C09129=1122.210,43.418,-53.082,179.810,7.126,149.381
C09130=1122.214,43.168,-53.066,179.809,7.121,149.380
C09131=1122.220,42.919,-53.051,179.808,7.117,149.380
C09132=1122.225,42.670,-53.035,179.807,7.113,149.379
C09133=1122.230,42.420,-53.019,179.806,7.109,149.379
C09134=1122.235,42.170,-53.004,179.805,7.105,149.378
C09135=1122.240,41.921,-52.989,179.804,7.101,149.377
C09136=1122.245,41.672,-52.973,179.803,7.097,149.377
C09137=1122.250,41.422,-52.956,179.802,7.093,149.376
C09138=1122.255,41.173,-52.941,179.800,7.088,149.376
C09139=1122.260,40.924,-52.926,179.799,7.084,149.375
C09140=1122.264,40.674,-52.910,179.798,7.080,149.374
C09141=1122.270,40.424,-52.894,179.797,7.076,149.374
C09142=1122.275,40.175,-52.879,179.796,7.072,149.373
C09143=1122.280,39.926,-52.864,179.795,7.067,149.373
C09144=1122.285,39.676,-52.848,179.794,7.063,149.372
C09145=1122.290,39.426,-52.832,179.792,7.059,149.371
C09146=1122.295,39.177,-52.817,179.791,7.055,149.371
C09147=1122.300,38.928,-52.802,179.790,7.050,149.370
C09148=1122.305,38.678,-52.786,179.789,7.046,149.369
C09149=1122.310,38.428,-52.771,179.788,7.042,149.369
C09150=1122.315,38.179,-52.755,179.786,7.038,149.368
C09151=1122.320,37.930,-52.739,179.785,7.034,149.368
C09152=1122.325,37.681,-52.724,179.784,7.029,149.367
C09153=1122.330,37.430,-52.708,179.783,7.025,149.366
C09154=1122.335,37.181,-52.693,179.783,7.021,149.366
C09155=1122.340,36.932,-52.678,179.781,7.018,149.365
C09156=1122.345,36.682,-52.663,179.780,7.013,149.365
C09157=1122.350,36.433,-52.648,179.779,7.009,149.364
C09158=1122.356,36.183,-52.632,179.778,7.005,149.363
C09159=1122.360,35.933,-52.616,179.777,7.000,149.363
C09160=1122.365,35.684,-52.601,179.776,6.996,149.362
C09161=1122.370,35.469,-52.588,179.774,6.992,149.362
C09162=1122.374,35.254,-52.575,179.774,6.989,149.361
C09163=1122.378,35.040,-52.562,179.773,6.985,149.361
C09164=1122.383,34.825,-52.549,179.772,6.981,149.360
C09165=1122.387,34.609,-52.535,179.771,6.978,149.360
C09166=1122.391,34.395,-52.523,179.770,6.974,149.359
C09167=1122.395,34.180,-52.509,179.769,6.970,149.358
C09168=1122.400,33.966,-52.496,179.768,6.966,149.358
C09169=1122.405,33.716,-52.481,179.767,6.962,149.357
C09170=1122.410,33.466,-52.466,179.766,6.958,149.357
C09171=1122.416,33.217,-52.451,179.765,6.954,149.356
C09172=1122.420,32.967,-52.436,179.764,6.950,149.355
C09173=1122.425,32.718,-52.420,179.763,6.946,149.355
C09174=1122.430,32.468,-52.406,179.762,6.941,149.354
C09175=1122.435,32.219,-52.390,179.760,6.937,149.353
C09176=1122.440,31.970,-52.375,179.759,6.933,149.353
C09177=1122.446,31.720,-52.360,179.758,6.929,149.352
C09178=1122.450,31.470,-52.345,179.757,6.924,149.352
C09179=1122.455,31.221,-52.330,179.756,6.920,149.351
C09180=1122.461,30.971,-52.315,179.755,6.916,149.350
C09181=1122.465,30.722,-52.300,179.754,6.911,149.350
C09182=1122.470,30.472,-52.284,179.753,6.907,149.349
C09183=1122.475,30.222,-52.270,179.752,6.903,149.348
C09184=1122.480,29.973,-52.255,179.751,6.898,149.348
C09185=1122.485,29.724,-52.240,179.750,6.894,149.347
C09186=1122.490,29.474,-52.225,179.749,6.890,149.346
C09187=1122.495,29.225,-52.210,179.748,6.885,149.346
C09188=1122.500,28.975,-52.195,179.747,6.881,149.345
C09189=1122.506,28.726,-52.180,179.746,6.876,149.344
C09190=1122.511,28.476,-52.166,179.745,6.872,149.344
C09191=1122.515,28.227,-52.151,179.744,6.868,149.343
C09192=1122.521,27.978,-52.135,179.743,6.863,149.342
C09193=1122.526,27.728,-52.121,179.742,6.859,149.342
C09194=1122.530,27.479,-52.106,179.741,6.855,149.341
C09195=1122.536,27.229,-52.091,179.740,6.850,149.340
C09196=1122.541,26.980,-52.076,179.739,6.846,149.340
C09197=1122.546,26.730,-52.062,179.738,6.842,149.339
C09198=1122.551,26.481,-52.046,179.737,6.838,149.338
C09199=1122.556,26.231,-52.032,179.736,6.833,149.337
C09200=1122.561,25.981,-52.017,179.735,6.829,149.337
C09201=1122.566,25.732,-52.002,179.734,6.824,149.336
C09202=1122.571,25.482,-51.988,179.733,6.820,149.335
C09203=1122.576,25.233,-51.973,179.732,6.816,149.335
C09204=1122.581,24.983,-51.958,179.731,6.811,149.334
C09205=1122.586,24.734,-51.943,179.730,6.807,149.334
C09206=1122.591,24.484,-51.928,179.729,6.802,149.333
C09207=1122.596,24.234,-51.914,179.728,6.798,149.332
C09208=1122.602,23.985,-51.899,179.727,6.794,149.331
C09209=1122.607,23.735,-51.884,179.726,6.789,149.331
C09210=1122.611,23.486,-51.870,179.725,6.785,149.330
C09211=1122.617,23.237,-51.855,179.724,6.780,149.329
C09212=1122.622,22.987,-51.841,179.723,6.776,149.329
C09213=1122.627,22.737,-51.826,179.722,6.772,149.328
C09214=1122.632,22.488,-51.811,179.721,6.767,149.327
C09215=1122.637,22.239,-51.797,179.721,6.763,149.326
C09216=1122.642,21.989,-51.783,179.720,6.758,149.326
C09217=1122.647,21.774,-51.770,179.719,6.754,149.325
C09218=1122.650,21.559,-51.757,179.718,6.751,149.325
C09219=1122.655,21.344,-51.745,179.717,6.747,149.324
C09220=1122.659,21.129,-51.733,179.716,6.743,149.323
C09221=1122.664,20.914,-51.720,179.715,6.739,149.323
C09222=1122.668,20.699,-51.707,179.715,6.735,149.322
C09223=1122.673,20.484,-51.695,179.714,6.731,149.321
C09224=1122.676,20.269,-51.683,179.713,6.728,149.321
C09225=1122.682,20.019,-51.668,179.712,6.723,149.320
C09226=1122.687,19.770,-51.653,179.711,6.719,149.319
C09227=1122.692,19.521,-51.639,179.710,6.714,149.319
C09228=1122.697,19.271,-51.624,179.710,6.710,149.318
C09229=1122.702,19.022,-51.610,179.709,6.705,149.317
C09230=1122.707,18.772,-51.596,179.707,6.700,149.317
C09231=1122.712,18.522,-51.582,179.706,6.695,149.316
C09232=1122.717,18.273,-51.567,179.705,6.691,149.315
C09233=1122.722,18.023,-51.553,179.705,6.686,149.314
C09234=1122.727,17.775,-51.538,179.704,6.682,149.313
C09235=1122.733,17.524,-51.524,179.703,6.678,149.313
C09236=1122.738,17.275,-51.509,179.702,6.673,149.312
C09237=1122.743,17.025,-51.495,179.701,6.669,149.311
C09238=1122.748,16.775,-51.481,179.700,6.664,149.310
C09239=1122.753,16.526,-51.467,179.699,6.660,149.310
C09240=1122.758,16.277,-51.453,179.698,6.655,149.309
C09241=1122.763,16.027,-51.438,179.698,6.651,149.308
C09242=1122.768,15.777,-51.424,179.697,6.646,149.308
C09243=1122.773,15.527,-51.410,179.696,6.642,149.307
C09244=1122.779,15.278,-51.396,179.695,6.637,149.306
C09245=1122.784,15.029,-51.382,179.695,6.633,149.305
C09246=1122.789,14.779,-51.367,179.693,6.628,149.305
C09247=1122.794,14.529,-51.353,179.692,6.623,149.304
C09248=1122.799,14.280,-51.339,179.691,6.618,149.303
C09249=1122.804,14.031,-51.325,179.691,6.614,149.302
C09250=1122.809,13.781,-51.311,179.690,6.609,149.301
C09251=1122.813,13.532,-51.297,179.689,6.605,149.301
C09252=1122.819,13.283,-51.283,179.688,6.600,149.300
C09253=1122.824,13.033,-51.269,179.688,6.596,149.299
C09254=1122.829,12.783,-51.254,179.687,6.591,149.298
C09255=1122.834,12.533,-51.240,179.686,6.587,149.298
C09256=1122.840,12.284,-51.227,179.686,6.582,149.297
C09257=1122.845,12.034,-51.213,179.684,6.577,149.296
C09258=1122.850,11.784,-51.198,179.683,6.572,149.295
C09259=1122.855,11.535,-51.184,179.682,6.568,149.294
C09260=1122.860,11.286,-51.170,179.682,6.563,149.294
C09261=1122.865,11.036,-51.156,179.681,6.558,149.293
C09262=1122.870,10.787,-51.143,179.680,6.554,149.292
C09263=1122.875,10.537,-51.129,179.680,6.549,149.291
C09264=1122.880,10.287,-51.115,179.679,6.545,149.291
C09265=1122.885,10.037,-51.100,179.678,6.540,149.290
C09266=1122.891,9.788,-51.087,179.678,6.536,149.289
C09267=1122.895,9.539,-51.072,179.676,6.530,149.288
C09268=1122.900,9.289,-51.059,179.675,6.526,149.287
C09269=1122.906,9.040,-51.045,179.675,6.521,149.286
C09270=1122.911,8.790,-51.031,179.674,6.516,149.286
C09271=1122.916,8.541,-51.017,179.673,6.512,149.285
C09272=1122.921,8.291,-51.004,179.673,6.507,149.284
C09273=1122.925,8.076,-50.991,179.672,6.504,149.283
C09274=1122.929,7.861,-50.980,179.672,6.499,149.282
C09275=1122.934,7.645,-50.968,179.671,6.495,149.282
C09276=1122.939,7.431,-50.956,179.671,6.492,149.281
C09277=1122.943,7.215,-50.944,179.670,6.487,149.280
C09278=1122.947,7.000,-50.933,179.670,6.484,149.280
C09279=1122.951,6.785,-50.920,179.670,6.480,149.279
C09280=1122.956,6.571,-50.909,179.670,6.476,149.278
C09281=1122.961,6.321,-50.895,179.669,6.471,149.277
C09282=1122.966,6.071,-50.881,179.669,6.467,149.276
C09283=1122.972,5.822,-50.867,179.668,6.462,149.275
C09284=1122.976,5.572,-50.854,179.667,6.458,149.275
C09285=1122.982,5.323,-50.840,179.667,6.454,149.274
C09286=1122.987,5.073,-50.826,179.667,6.449,149.273
C09287=1122.992,4.823,-50.812,179.666,6.444,149.272
C09288=1122.997,4.574,-50.799,179.665,6.440,149.271
C09289=1123.002,4.324,-50.786,179.665,6.435,149.270
C09290=1123.008,4.075,-50.772,179.664,6.430,149.269
C09291=1123.012,3.825,-50.758,179.664,6.427,149.269
C09292=1123.018,3.576,-50.745,179.663,6.422,149.268
C09293=1123.023,3.326,-50.730,179.663,6.417,149.267
C09294=1123.027,3.076,-50.718,179.662,6.412,149.266
C09295=1123.033,2.827,-50.704,179.662,6.408,149.265
C09296=1123.038,2.577,-50.690,179.661,6.404,149.265
C09297=1123.043,2.328,-50.677,179.661,6.400,149.264
C09298=1123.048,2.078,-50.663,179.660,6.395,149.263
C09299=1123.054,1.829,-50.649,179.660,6.390,149.262
C09300=1123.058,1.579,-50.636,179.659,6.385,149.261
C09301=1123.064,1.330,-50.622,179.658,6.381,149.260
C09302=1123.068,1.080,-50.609,179.658,6.377,149.260
C09303=1123.074,0.831,-50.595,179.658,6.372,149.259
C09304=1123.079,0.580,-50.582,179.657,6.368,149.258
C09305=1123.084,0.331,-50.569,179.656,6.363,149.257
C09306=1123.089,0.081,-50.555,179.656,6.359,149.256
C09307=1123.094,-0.168,-50.542,179.655,6.354,149.255
C09308=1123.099,-0.418,-50.528,179.655,6.349,149.254
C09309=1123.104,-0.667,-50.516,179.654,6.346,149.254
C09310=1123.110,-0.917,-50.502,179.654,6.341,149.253
C09311=1123.115,-1.166,-50.488,179.653,6.336,149.252
C09312=1123.120,-1.417,-50.475,179.652,6.332,149.251
C09313=1123.125,-1.666,-50.461,179.652,6.327,149.250
C09314=1123.130,-1.916,-50.448,179.651,6.322,149.250
C09315=1123.136,-2.165,-50.435,179.651,6.318,149.249
C09316=1123.140,-2.415,-50.421,179.650,6.314,149.248
C09317=1123.146,-2.664,-50.408,179.650,6.309,149.247
C09318=1123.150,-2.914,-50.395,179.649,6.305,149.246
C09319=1123.156,-3.163,-50.381,179.648,6.300,149.246
C09320=1123.161,-3.413,-50.369,179.648,6.296,149.245
C09321=1123.166,-3.663,-50.355,179.647,6.291,149.244
C09322=1123.171,-3.912,-50.343,179.647,6.286,149.243
C09323=1123.176,-4.162,-50.328,179.646,6.282,149.242
C09324=1123.181,-4.411,-50.316,179.645,6.277,149.241
C09325=1123.187,-4.661,-50.302,179.645,6.273,149.241
C09326=1123.192,-4.911,-50.289,179.644,6.269,149.240
C09327=1123.197,-5.160,-50.276,179.644,6.264,149.239
C09328=1123.202,-5.410,-50.263,179.643,6.259,149.238
C09329=1123.207,-5.624,-50.251,179.642,6.255,149.237
C09330=1123.211,-5.840,-50.240,179.642,6.251,149.237
C09331=1123.215,-6.056,-50.229,179.641,6.248,149.236
C09332=1123.220,-6.270,-50.217,179.640,6.244,149.235
C09333=1123.225,-6.486,-50.206,179.641,6.240,149.235
C09334=1123.229,-6.701,-50.195,179.640,6.236,149.234
C09335=1123.234,-6.916,-50.183,179.639,6.232,149.233
C09336=1123.237,-7.131,-50.172,179.639,6.228,149.233
C09337=1123.243,-7.380,-50.159,179.638,6.224,149.232
C09338=1123.248,-7.630,-50.146,179.637,6.219,149.231
C09339=1123.253,-7.880,-50.133,179.637,6.214,149.230
C09340=1123.258,-8.129,-50.120,179.636,6.210,149.229
C09341=1123.263,-8.379,-50.107,179.635,6.205,149.229
C09342=1123.269,-8.629,-50.094,179.635,6.201,149.228
C09343=1123.274,-8.878,-50.082,179.634,6.196,149.227
C09344=1123.278,-9.128,-50.069,179.633,6.192,149.226
C09345=1123.284,-9.377,-50.055,179.633,6.187,149.225
C09346=1123.289,-9.627,-50.042,179.632,6.182,149.224
C09347=1123.294,-9.877,-50.029,179.631,6.178,149.224
C09348=1123.299,-10.126,-50.016,179.631,6.173,149.223
C09349=1123.305,-10.376,-50.003,179.630,6.168,149.222
C09350=1123.310,-10.625,-49.991,179.630,6.164,149.221
C09351=1123.314,-10.875,-49.978,179.629,6.159,149.220
C09352=1123.320,-11.125,-49.965,179.628,6.155,149.219
C09353=1123.325,-11.374,-49.952,179.628,6.150,149.219
C09354=1123.330,-11.624,-49.939,179.627,6.145,149.218
C09355=1123.336,-11.874,-49.926,179.626,6.141,149.217
C09356=1123.341,-12.123,-49.913,179.626,6.136,149.216
C09357=1123.345,-12.373,-49.900,179.625,6.132,149.215
C09358=1123.350,-12.622,-49.888,179.624,6.127,149.215
C09359=1123.356,-12.872,-49.876,179.624,6.122,149.214
C09360=1123.362,-13.122,-49.863,179.623,6.118,149.213
C09361=1123.366,-13.372,-49.850,179.622,6.113,149.212
C09362=1123.371,-13.621,-49.837,179.622,6.108,149.211
C09363=1123.376,-13.870,-49.824,179.621,6.104,149.211
C09364=1123.382,-14.120,-49.811,179.620,6.099,149.210
C09365=1123.387,-14.370,-49.798,179.620,6.095,149.209
C09366=1123.392,-14.619,-49.786,179.619,6.090,149.208
C09367=1123.397,-14.869,-49.773,179.618,6.086,149.207
C09368=1123.402,-15.119,-49.761,179.618,6.081,149.206
C09369=1123.408,-15.368,-49.749,179.617,6.076,149.206
C09370=1123.413,-15.618,-49.735,179.616,6.072,149.205
C09371=1123.418,-15.868,-49.722,179.615,6.066,149.204
C09372=1123.423,-16.117,-49.710,179.615,6.061,149.203
C09373=1123.429,-16.367,-49.698,179.614,6.057,149.202
C09374=1123.434,-16.616,-49.685,179.613,6.052,149.201
C09375=1123.438,-16.866,-49.672,179.613,6.048,149.201
C09376=1123.443,-17.116,-49.660,179.612,6.043,149.200
C09377=1123.449,-17.365,-49.647,179.611,6.039,149.199
C09378=1123.455,-17.615,-49.635,179.611,6.034,149.198
C09379=1123.460,-17.864,-49.622,179.610,6.029,149.197
C09380=1123.464,-18.114,-49.609,179.609,6.024,149.197
C09381=1123.470,-18.364,-49.597,179.608,6.019,149.196
C09382=1123.475,-18.614,-49.585,179.608,6.014,149.195
C09383=1123.480,-18.863,-49.572,179.607,6.010,149.194
C09384=1123.485,-19.112,-49.559,179.606,6.005,149.193
C09385=1123.490,-19.328,-49.548,179.606,6.001,149.192
C09386=1123.494,-19.543,-49.538,179.605,5.997,149.192
C09387=1123.499,-19.758,-49.528,179.605,5.993,149.191
C09388=1123.503,-19.974,-49.517,179.604,5.989,149.190
C09389=1123.507,-20.188,-49.506,179.604,5.984,149.189
C09390=1123.512,-20.404,-49.495,179.603,5.980,149.189
C09391=1123.517,-20.620,-49.485,179.602,5.977,149.188
C09392=1123.521,-20.835,-49.474,179.601,5.972,149.187
C09393=1123.526,-21.084,-49.462,179.601,5.968,149.187
C09394=1123.531,-21.334,-49.450,179.600,5.963,149.186
C09395=1123.536,-21.584,-49.437,179.599,5.957,149.185
C09396=1123.542,-21.833,-49.424,179.599,5.953,149.184
C09397=1123.547,-22.083,-49.413,179.598,5.948,149.183
C09398=1123.552,-22.332,-49.400,179.597,5.943,149.182
C09399=1123.558,-22.582,-49.388,179.597,5.939,149.181
C09400=1123.563,-22.831,-49.376,179.596,5.933,149.181
C09401=1123.568,-23.081,-49.364,179.595,5.928,149.180
C09402=1123.573,-23.331,-49.351,179.594,5.924,149.179
C09403=1123.578,-23.581,-49.339,179.594,5.919,149.178
C09404=1123.583,-23.831,-49.326,179.593,5.914,149.177
C09405=1123.589,-24.081,-49.314,179.592,5.909,149.176
C09406=1123.594,-24.330,-49.302,179.592,5.904,149.175
C09407=1123.599,-24.580,-49.290,179.591,5.899,149.175
C09408=1123.604,-24.829,-49.277,179.590,5.894,149.174
C09409=1123.609,-25.079,-49.266,179.589,5.890,149.173
C09410=1123.614,-25.329,-49.254,179.589,5.885,149.172
C09411=1123.619,-25.578,-49.241,179.588,5.879,149.171
C09412=1123.625,-25.828,-49.230,179.587,5.875,149.170
C09413=1123.630,-26.077,-49.217,179.587,5.870,149.169
C09414=1123.635,-26.327,-49.205,179.589,5.866,149.168
C09415=1123.641,-26.577,-49.193,179.589,5.862,149.167
C09416=1123.645,-26.826,-49.181,179.590,5.858,149.166
C09417=1123.651,-27.076,-49.169,179.591,5.854,149.165
C09418=1123.656,-27.325,-49.157,179.591,5.850,149.164
C09419=1123.661,-27.575,-49.145,179.592,5.846,149.163
C09420=1123.667,-27.825,-49.133,179.593,5.842,149.161
C09421=1123.672,-28.075,-49.120,179.594,5.838,149.160
C09422=1123.677,-28.324,-49.109,179.594,5.834,149.159
C09423=1123.682,-28.574,-49.097,179.594,5.829,149.158
C09424=1123.687,-28.824,-49.085,179.596,5.826,149.157
C09425=1123.693,-29.073,-49.073,179.596,5.822,149.156
C09426=1123.698,-29.323,-49.061,179.596,5.818,149.155
C09427=1123.702,-29.572,-49.049,179.597,5.814,149.154
C09428=1123.708,-29.822,-49.037,179.597,5.810,149.153
C09429=1123.713,-30.072,-49.025,179.597,5.805,149.152
C09430=1123.718,-30.322,-49.012,179.597,5.801,149.151
C09431=1123.724,-30.572,-49.001,179.597,5.797,149.150
C09432=1123.728,-30.821,-48.989,179.598,5.792,149.149
C09433=1123.734,-31.070,-48.978,179.598,5.788,149.148
C09434=1123.740,-31.320,-48.965,179.597,5.784,149.147
C09435=1123.745,-31.570,-48.953,179.597,5.780,149.147
C09436=1123.750,-31.819,-48.942,179.597,5.775,149.146
C09437=1123.755,-32.069,-48.929,179.597,5.771,149.145
C09438=1123.760,-32.319,-48.917,179.597,5.767,149.144
C09439=1123.766,-32.568,-48.906,179.597,5.762,149.143
C09440=1123.770,-32.818,-48.894,179.596,5.758,149.142
C09441=1123.775,-33.033,-48.884,179.596,5.754,149.141
C09442=1123.779,-33.249,-48.873,179.596,5.750,149.140
C09443=1123.784,-33.464,-48.863,179.596,5.747,149.140
C09444=1123.789,-33.679,-48.853,179.596,5.743,149.139
C09445=1123.793,-33.895,-48.843,179.595,5.738,149.138
C09446=1123.798,-34.110,-48.832,179.595,5.735,149.138
C09447=1123.802,-34.325,-48.822,179.594,5.731,149.137
C09448=1123.806,-34.541,-48.812,179.594,5.726,149.136
C09449=1123.812,-34.790,-48.801,179.594,5.723,149.135
C09450=1123.817,-35.040,-48.789,179.593,5.718,149.134
C09451=1123.823,-35.290,-48.777,179.593,5.713,149.133
C09452=1123.827,-35.539,-48.765,179.591,5.708,149.133
C09453=1123.833,-35.789,-48.754,179.591,5.703,149.132
C09454=1123.838,-36.039,-48.742,179.590,5.699,149.131
C09455=1123.843,-36.288,-48.730,179.589,5.694,149.130
C09456=1123.848,-36.538,-48.718,179.589,5.690,149.129
C09457=1123.854,-36.788,-48.706,179.587,5.684,149.129
C09458=1123.859,-37.037,-48.695,179.587,5.680,149.128
C09459=1123.864,-37.287,-48.683,179.585,5.675,149.127
C09460=1123.869,-37.537,-48.672,179.585,5.670,149.126
C09461=1123.874,-37.787,-48.660,179.583,5.665,149.126
C09462=1123.880,-38.037,-48.648,179.583,5.660,149.125
C09463=1123.885,-38.286,-48.637,179.581,5.655,149.124
C09464=1123.890,-38.535,-48.625,179.580,5.650,149.123
C09465=1123.895,-38.785,-48.614,179.579,5.645,149.122
C09466=1123.901,-39.035,-48.602,179.578,5.640,149.122
C09467=1123.905,-39.285,-48.591,179.577,5.634,149.121
C09468=1123.911,-39.534,-48.579,179.575,5.629,149.120
C09469=1123.917,-39.784,-48.567,179.574,5.624,149.120
C09470=1123.921,-40.033,-48.556,179.573,5.618,149.119
C09471=1123.927,-40.283,-48.544,179.571,5.613,149.118
C09472=1123.932,-40.533,-48.533,179.570,5.608,149.117
C09473=1123.938,-40.783,-48.522,179.569,5.602,149.116
C09474=1123.943,-41.032,-48.511,179.567,5.597,149.116
C09475=1123.948,-41.282,-48.499,179.565,5.592,149.115
C09476=1123.953,-41.531,-48.488,179.564,5.586,149.114
C09477=1123.959,-41.781,-48.476,179.562,5.581,149.114
C09478=1123.963,-42.031,-48.465,179.560,5.575,149.113
C09479=1123.969,-42.281,-48.454,179.559,5.569,149.112
C09480=1123.974,-42.530,-48.443,179.557,5.563,149.111
C09481=1123.979,-42.780,-48.431,179.555,5.558,149.111
C09482=1123.985,-43.030,-48.420,179.554,5.552,149.110
C09483=1123.990,-43.279,-48.409,179.553,5.547,149.109
C09484=1123.996,-43.529,-48.397,179.553,5.542,149.108
C09485=1124.000,-43.779,-48.386,179.554,5.538,149.107
C09486=1124.005,-44.029,-48.375,179.554,5.533,149.106
C09487=1124.011,-44.279,-48.364,179.554,5.528,149.105
C09488=1124.016,-44.528,-48.353,179.554,5.523,149.103
C09489=1124.021,-44.778,-48.342,179.554,5.518,149.103
C09490=1124.027,-45.027,-48.330,179.555,5.514,149.101
C09491=1124.032,-45.277,-48.319,179.555,5.509,149.100
C09492=1124.037,-45.527,-48.308,179.555,5.505,149.099
C09493=1124.042,-45.776,-48.297,179.555,5.500,149.098
C09494=1124.047,-46.026,-48.286,179.555,5.495,149.097
C09495=1124.053,-46.276,-48.274,179.556,5.490,149.096
C09496=1124.058,-46.525,-48.263,179.555,5.486,149.095
C09497=1124.063,-46.741,-48.254,179.556,5.481,149.094
C09498=1124.067,-46.956,-48.245,179.556,5.477,149.093
C09499=1124.072,-47.172,-48.235,179.556,5.473,149.092
C09500=1124.076,-47.387,-48.225,179.556,5.469,149.091
C09501=1124.081,-47.603,-48.216,179.557,5.465,149.090
C09502=1124.085,-47.818,-48.206,179.557,5.461,149.089
C09503=1124.090,-48.034,-48.197,179.557,5.458,149.088
C09504=1124.094,-48.249,-48.187,179.557,5.454,149.087
C09505=1124.100,-48.499,-48.176,179.557,5.448,149.086
C09506=1124.105,-48.748,-48.165,179.557,5.444,149.085
C09507=1124.110,-48.998,-48.154,179.557,5.439,149.084
C09508=1124.115,-49.247,-48.144,179.558,5.434,149.083
C09509=1124.121,-49.497,-48.132,179.558,5.430,149.082
C09510=1124.126,-49.747,-48.121,179.558,5.425,149.081
C09511=1124.131,-49.996,-48.110,179.558,5.420,149.080
C09512=1124.137,-50.247,-48.099,179.559,5.416,149.079
C09513=1124.142,-50.496,-48.088,179.558,5.411,149.078
C09514=1124.147,-50.746,-48.077,179.559,5.406,149.077
C09515=1124.152,-50.996,-48.066,179.559,5.401,149.076
C09516=1124.158,-51.246,-48.055,179.559,5.397,149.075
C09517=1124.163,-51.495,-48.044,179.559,5.392,149.073
C09518=1124.169,-51.745,-48.034,179.559,5.387,149.072
C09519=1124.173,-51.994,-48.023,179.560,5.383,149.071
C09520=1124.179,-52.244,-48.012,179.560,5.378,149.070
C09521=1124.184,-52.494,-48.000,179.560,5.374,149.069
C09522=1124.189,-52.744,-47.990,179.560,5.369,149.068
C09523=1124.195,-52.993,-47.979,179.560,5.365,149.067
C09524=1124.200,-53.243,-47.968,179.561,5.359,149.066
C09525=1124.205,-53.493,-47.958,179.561,5.354,149.065
C09526=1124.211,-53.743,-47.946,179.561,5.350,149.064
C09527=1124.216,-53.992,-47.936,179.561,5.345,149.063
C09528=1124.221,-54.242,-47.925,179.562,5.341,149.062
C09529=1124.226,-54.491,-47.915,179.561,5.336,149.061
C09530=1124.231,-54.741,-47.903,179.562,5.332,149.060
C09531=1124.237,-54.991,-47.893,179.562,5.327,149.058
C09532=1124.242,-55.241,-47.883,179.562,5.322,149.057
C09533=1124.248,-55.490,-47.871,179.562,5.317,149.056
C09534=1124.253,-55.740,-47.860,179.562,5.312,149.055
C09535=1124.258,-55.990,-47.850,179.563,5.308,149.054
C09536=1124.263,-56.240,-47.839,179.563,5.303,149.053
C09537=1124.268,-56.490,-47.828,179.563,5.299,149.052
C09538=1124.273,-56.739,-47.817,179.563,5.294,149.051
C09539=1124.278,-56.989,-47.807,179.564,5.290,149.050
C09540=1124.284,-57.238,-47.797,179.564,5.285,149.049
C09541=1124.289,-57.488,-47.785,179.563,5.280,149.048
C09542=1124.294,-57.738,-47.775,179.564,5.276,149.047
C09543=1124.301,-57.988,-47.764,179.564,5.270,149.045
C09544=1124.306,-58.238,-47.754,179.564,5.266,149.045
C09545=1124.311,-58.487,-47.743,179.564,5.261,149.043
C09546=1124.316,-58.737,-47.732,179.565,5.257,149.042
C09547=1124.321,-58.986,-47.722,179.565,5.252,149.041
C09548=1124.326,-59.236,-47.711,179.565,5.248,149.040
C09549=1124.332,-59.486,-47.701,179.565,5.243,149.039
C09550=1124.337,-59.736,-47.690,179.565,5.238,149.038
C09551=1124.342,-59.985,-47.680,179.566,5.234,149.037
C09552=1124.347,-60.235,-47.669,179.565,5.229,149.036
C09553=1124.352,-60.451,-47.659,179.565,5.224,149.035
C09554=1124.357,-60.667,-47.651,179.564,5.220,149.034
C09555=1124.361,-60.882,-47.642,179.563,5.215,149.034
C09556=1124.365,-61.097,-47.633,179.563,5.211,149.033
C09557=1124.370,-61.313,-47.623,179.562,5.206,149.032
C09558=1124.374,-61.528,-47.614,179.561,5.202,149.031
C09559=1124.379,-61.744,-47.605,179.561,5.197,149.031
C09560=1124.383,-61.959,-47.596,179.560,5.193,149.030
C09561=1124.389,-62.209,-47.586,179.559,5.187,149.029
C09562=1124.394,-62.458,-47.576,179.558,5.182,149.028
C09563=1124.399,-62.708,-47.565,179.557,5.177,149.027
C09564=1124.405,-62.958,-47.555,179.556,5.171,149.026
C09565=1124.410,-63.208,-47.544,179.556,5.166,149.025
C09566=1124.415,-63.458,-47.534,179.555,5.161,149.024
C09567=1124.421,-63.707,-47.524,179.554,5.155,149.023
C09568=1124.426,-63.957,-47.513,179.554,5.150,149.022
C09569=1124.431,-64.206,-47.502,179.553,5.145,149.021
C09570=1124.437,-64.456,-47.492,179.553,5.140,149.021
C09571=1124.442,-64.706,-47.482,179.552,5.134,149.020
C09572=1124.448,-64.956,-47.471,179.551,5.129,149.019
C09573=1124.453,-65.205,-47.461,179.551,5.124,149.018
C09574=1124.457,-65.455,-47.451,179.550,5.118,149.017
C09575=1124.463,-65.705,-47.441,179.550,5.113,149.016
C09576=1124.469,-65.954,-47.431,179.549,5.108,149.015
C09577=1124.474,-66.204,-47.420,179.548,5.103,149.014
C09578=1124.479,-66.454,-47.410,179.548,5.097,149.013
C09579=1124.485,-66.704,-47.400,179.547,5.091,149.012
C09580=1124.489,-66.954,-47.390,179.546,5.087,149.011
C09581=1124.495,-67.204,-47.380,179.546,5.081,149.010
C09582=1124.501,-67.453,-47.370,179.546,5.076,149.009
C09583=1124.506,-67.703,-47.360,179.545,5.070,149.008
C09584=1124.511,-67.953,-47.349,179.545,5.065,149.007
C09585=1124.517,-68.203,-47.339,179.544,5.060,149.006
C09586=1124.522,-68.452,-47.330,179.544,5.054,149.005
C09587=1124.527,-68.702,-47.319,179.544,5.050,149.004
C09588=1124.532,-68.952,-47.309,179.543,5.044,149.003
C09589=1124.538,-69.201,-47.299,179.543,5.039,149.002
C09590=1124.543,-69.451,-47.290,179.542,5.033,149.001
C09591=1124.548,-69.701,-47.279,179.542,5.028,149.000
C09592=1124.554,-69.951,-47.269,179.541,5.023,148.999
C09593=1124.559,-70.200,-47.259,179.541,5.018,148.998
C09594=1124.564,-70.450,-47.249,179.541,5.013,148.997
C09595=1124.570,-70.700,-47.240,179.540,5.007,148.995
C09596=1124.575,-70.950,-47.229,179.540,5.002,148.994
C09597=1124.581,-71.199,-47.219,179.539,4.996,148.993
C09598=1124.585,-71.449,-47.209,179.540,4.991,148.992
C09599=1124.591,-71.699,-47.200,179.539,4.986,148.991
C09600=1124.596,-71.949,-47.189,179.539,4.980,148.990
C09601=1124.601,-72.198,-47.179,179.539,4.975,148.989
C09602=1124.607,-72.448,-47.169,179.539,4.970,148.988
C09603=1124.613,-72.698,-47.160,179.538,4.964,148.987
C09604=1124.617,-72.947,-47.150,179.538,4.959,148.986
C09605=1124.623,-73.197,-47.140,179.538,4.954,148.985
C09606=1124.628,-73.448,-47.130,179.537,4.948,148.984
C09607=1124.633,-73.697,-47.120,179.538,4.943,148.982
C09608=1124.639,-73.946,-47.110,179.538,4.938,148.981
C09609=1124.643,-74.162,-47.102,179.537,4.933,148.980
C09610=1124.649,-74.378,-47.094,179.538,4.929,148.979
C09611=1124.653,-74.593,-47.085,179.537,4.925,148.979
C09612=1124.657,-74.809,-47.077,179.537,4.920,148.978
C09613=1124.662,-75.025,-47.068,179.537,4.916,148.977
C09614=1124.666,-75.240,-47.060,179.537,4.911,148.976
C09615=1124.671,-75.455,-47.052,179.536,4.906,148.975
C09616=1124.676,-75.671,-47.043,179.537,4.902,148.974
C09617=1124.682,-75.921,-47.033,179.536,4.896,148.973
C09618=1124.687,-76.170,-47.024,179.536,4.891,148.972
C09619=1124.692,-76.420,-47.014,179.536,4.886,148.970
C09620=1124.697,-76.670,-47.004,179.537,4.881,148.969
C09621=1124.703,-76.921,-46.995,179.537,4.876,148.968
C09622=1124.707,-77.170,-46.985,179.537,4.871,148.967
C09623=1124.713,-77.420,-46.975,179.537,4.865,148.966
C09624=1124.719,-77.669,-46.965,179.536,4.860,148.965
C09625=1124.724,-77.919,-46.956,179.536,4.855,148.964
C09626=1124.730,-78.169,-46.946,179.536,4.850,148.963
C09627=1124.735,-78.419,-46.937,179.537,4.844,148.961
C09628=1124.741,-78.668,-46.927,179.537,4.839,148.960
C09629=1124.746,-78.918,-46.918,179.537,4.834,148.959
C09630=1124.751,-79.168,-46.908,179.537,4.829,148.958
C09631=1124.756,-79.417,-46.899,179.537,4.824,148.957
C09632=1124.762,-79.667,-46.889,179.537,4.819,148.956
C09633=1124.767,-79.917,-46.880,179.538,4.813,148.954
C09634=1124.773,-80.166,-46.870,179.538,4.808,148.953
C09635=1124.777,-80.417,-46.860,179.538,4.803,148.952
C09636=1124.783,-80.667,-46.851,179.538,4.798,148.951
C09637=1124.788,-80.916,-46.841,179.538,4.793,148.950
C09638=1124.794,-81.167,-46.832,179.538,4.788,148.949
C09639=1124.799,-81.416,-46.822,179.539,4.782,148.947
C09640=1124.804,-81.666,-46.813,179.539,4.777,148.946
C09641=1124.810,-81.916,-46.804,179.539,4.772,148.945
C09642=1124.815,-82.165,-46.794,179.539,4.767,148.944
C09643=1124.821,-82.415,-46.785,179.539,4.762,148.943
C09644=1124.826,-82.664,-46.775,179.539,4.757,148.941
C09645=1124.832,-82.915,-46.766,179.540,4.752,148.940
C09646=1124.837,-83.164,-46.757,179.541,4.747,148.939
C09647=1124.842,-83.414,-46.747,179.541,4.742,148.938
C09648=1124.847,-83.664,-46.738,179.541,4.736,148.937
C09649=1124.853,-83.914,-46.729,179.541,4.731,148.935
C09650=1124.858,-84.163,-46.719,179.542,4.726,148.934
C09651=1124.863,-84.413,-46.710,179.542,4.722,148.933
C09652=1124.869,-84.663,-46.701,179.542,4.717,148.932
C09653=1124.874,-84.913,-46.691,179.543,4.711,148.931
C09654=1124.879,-85.162,-46.682,179.543,4.706,148.929
C09655=1124.884,-85.412,-46.673,179.544,4.701,148.928
C09656=1124.890,-85.662,-46.663,179.544,4.696,148.927
C09657=1124.895,-85.912,-46.654,179.544,4.691,148.926
C09658=1124.900,-86.161,-46.645,179.545,4.686,148.925
C09659=1124.906,-86.412,-46.635,179.545,4.682,148.923
C09660=1124.912,-86.661,-46.627,179.546,4.676,148.922
C09661=1124.917,-86.910,-46.617,179.546,4.671,148.921
C09662=1124.923,-87.160,-46.608,179.546,4.666,148.920
C09663=1124.928,-87.410,-46.599,179.547,4.661,148.918
C09664=1124.933,-87.660,-46.590,179.547,4.656,148.917
C09665=1124.937,-87.876,-46.582,179.548,4.652,148.916
C09666=1124.942,-88.092,-46.573,179.548,4.648,148.915
C09667=1124.947,-88.307,-46.566,179.549,4.644,148.914
C09668=1124.951,-88.523,-46.558,179.550,4.640,148.913
C09669=1124.956,-88.738,-46.550,179.550,4.635,148.912
C09670=1124.961,-88.954,-46.541,179.551,4.631,148.911
C09671=1124.965,-89.170,-46.533,179.551,4.626,148.910
C09672=1124.970,-89.385,-46.527,179.551,4.622,148.909
C09673=1124.975,-89.635,-46.517,179.552,4.617,148.907
C09674=1124.981,-89.885,-46.507,179.552,4.612,148.906
C09675=1124.986,-90.135,-46.499,179.553,4.608,148.905
C09676=1124.992,-90.384,-46.490,179.553,4.603,148.904
C09677=1124.997,-90.634,-46.481,179.554,4.598,148.903
C09678=1125.003,-90.884,-46.471,179.555,4.593,148.901
C09679=1125.008,-91.134,-46.462,179.556,4.588,148.900
C09680=1125.013,-91.384,-46.453,179.557,4.584,148.899
C09681=1125.018,-91.633,-46.444,179.557,4.579,148.898
C09682=1125.024,-91.883,-46.435,179.558,4.574,148.896
C09683=1125.030,-92.133,-46.426,179.558,4.569,148.895
C09684=1125.035,-92.383,-46.417,179.559,4.565,148.894
C09685=1125.040,-92.632,-46.408,179.560,4.560,148.893
C09686=1125.045,-92.882,-46.399,179.560,4.555,148.891
C09687=1125.051,-93.132,-46.390,179.561,4.550,148.890
C09688=1125.056,-93.382,-46.381,179.562,4.546,148.889
C09689=1125.062,-93.631,-46.372,179.562,4.541,148.888
C09690=1125.067,-93.881,-46.363,179.564,4.536,148.886
C09691=1125.072,-94.131,-46.354,179.564,4.532,148.885
C09692=1125.078,-94.381,-46.345,179.565,4.527,148.884
C09693=1125.083,-94.631,-46.336,179.565,4.522,148.883
C09694=1125.088,-94.881,-46.327,179.566,4.517,148.882
C09695=1125.094,-95.131,-46.318,179.566,4.512,148.880
C09696=1125.099,-95.380,-46.310,179.567,4.508,148.879
C09697=1125.105,-95.630,-46.301,179.567,4.502,148.878
C09698=1125.110,-95.880,-46.291,179.567,4.497,148.877
C09699=1125.116,-96.130,-46.282,179.567,4.492,148.876
C09700=1125.121,-96.380,-46.274,179.568,4.488,148.874
C09701=1125.127,-96.629,-46.265,179.568,4.483,148.873
C09702=1125.132,-96.879,-46.256,179.568,4.477,148.872
C09703=1125.137,-97.129,-46.247,179.568,4.473,148.871
C09704=1125.142,-97.378,-46.238,179.568,4.467,148.870
C09705=1125.148,-97.629,-46.229,179.569,4.463,148.869
C09706=1125.153,-97.878,-46.220,179.569,4.458,148.868
C09707=1125.159,-98.128,-46.211,179.570,4.453,148.866
C09708=1125.164,-98.377,-46.202,179.570,4.448,148.865
C09709=1125.169,-98.627,-46.194,179.570,4.442,148.864
C09710=1125.174,-98.877,-46.185,179.570,4.437,148.863
C09711=1125.180,-99.126,-46.176,179.571,4.433,148.862
C09712=1125.185,-99.376,-46.167,179.571,4.428,148.860
C09713=1125.191,-99.627,-46.159,179.571,4.423,148.860
C09714=1125.196,-99.876,-46.150,179.571,4.418,148.858
C09715=1125.202,-100.126,-46.142,179.571,4.413,148.857
C09716=1125.208,-100.376,-46.132,179.572,4.407,148.856
C09717=1125.213,-100.626,-46.123,179.572,4.403,148.855
C09718=1125.218,-100.875,-46.114,179.573,4.398,148.854
C09719=1125.224,-101.125,-46.107,179.573,4.393,148.852
C09720=1125.229,-101.375,-46.098,179.573,4.388,148.851
C09721=1125.233,-101.591,-46.090,179.573,4.384,148.850
C09722=1125.239,-101.807,-46.083,179.573,4.379,148.849
C09723=1125.243,-102.022,-46.075,179.573,4.375,148.848
C09724=1125.248,-102.238,-46.068,179.574,4.370,148.847
C09725=1125.252,-102.454,-46.060,179.574,4.366,148.846
C09726=1125.257,-102.669,-46.052,179.574,4.362,148.845
C09727=1125.261,-102.885,-46.045,179.575,4.358,148.844
C09728=1125.266,-103.101,-46.037,179.575,4.353,148.843
C09729=1125.272,-103.351,-46.029,179.575,4.347,148.842
C09730=1125.277,-103.601,-46.020,179.575,4.343,148.841
C09731=1125.282,-103.851,-46.011,179.575,4.337,148.840
C09732=1125.288,-104.100,-46.003,179.576,4.333,148.839
C09733=1125.293,-104.350,-45.995,179.576,4.328,148.837
C09734=1125.298,-104.600,-45.986,179.576,4.323,148.836
C09735=1125.303,-104.849,-45.978,179.576,4.318,148.835
C09736=1125.309,-105.100,-45.970,179.577,4.312,148.834
C09737=1125.314,-105.349,-45.961,179.577,4.307,148.833
C09738=1125.320,-105.599,-45.952,179.577,4.302,148.831
C09739=1125.325,-105.849,-45.944,179.577,4.297,148.830
C09740=1125.330,-106.099,-45.935,179.577,4.292,148.829
C09741=1125.336,-106.348,-45.927,179.577,4.287,148.828
C09742=1125.342,-106.598,-45.918,179.578,4.282,148.827
C09743=1125.347,-106.848,-45.910,179.578,4.277,148.826
C09744=1125.353,-107.097,-45.901,179.578,4.271,148.825
C09745=1125.358,-107.348,-45.893,179.578,4.266,148.823
C09746=1125.363,-107.598,-45.884,179.579,4.261,148.822
C09747=1125.368,-107.847,-45.876,179.579,4.256,148.821
C09748=1125.374,-108.097,-45.868,179.579,4.251,148.820
C09749=1125.379,-108.347,-45.859,179.579,4.245,148.819
C09750=1125.385,-108.597,-45.851,179.580,4.240,148.817
C09751=1125.390,-108.847,-45.842,179.579,4.236,148.816
C09752=1125.395,-109.096,-45.833,179.580,4.230,148.815
C09753=1125.401,-109.346,-45.826,179.580,4.225,148.814
C09754=1125.406,-109.596,-45.817,179.580,4.220,148.813
C09755=1125.412,-109.846,-45.809,179.580,4.215,148.812
C09756=1125.417,-110.095,-45.800,179.581,4.210,148.810
C09757=1125.423,-110.346,-45.792,179.581,4.204,148.809
C09758=1125.428,-110.595,-45.784,179.581,4.199,148.808
C09759=1125.433,-110.845,-45.776,179.581,4.194,148.807
C09760=1125.439,-111.094,-45.768,179.582,4.189,148.806
C09761=1125.444,-111.345,-45.759,179.582,4.184,148.804
C09762=1125.450,-111.594,-45.751,179.582,4.179,148.803
C09763=1125.456,-111.844,-45.743,179.582,4.173,148.802
C09764=1125.460,-112.094,-45.734,179.583,4.168,148.801
C09765=1125.466,-112.344,-45.727,179.582,4.162,148.800
C09766=1125.471,-112.594,-45.718,179.582,4.157,148.799
C09767=1125.477,-112.843,-45.710,179.582,4.152,148.797
C09768=1125.482,-113.093,-45.701,179.582,4.147,148.796
C09769=1125.488,-113.343,-45.694,179.583,4.142,148.795
C09770=1125.493,-113.592,-45.685,179.583,4.137,148.794
C09771=1125.499,-113.842,-45.677,179.583,4.132,148.793
C09772=1125.504,-114.092,-45.670,179.584,4.126,148.791
C09773=1125.510,-114.342,-45.661,179.584,4.121,148.790
C09774=1125.515,-114.592,-45.653,179.583,4.115,148.789
C09775=1125.521,-114.843,-45.645,179.584,4.110,148.788
C09776=1125.526,-115.091,-45.637,179.584,4.105,148.787
C09777=1125.531,-115.307,-45.630,179.584,4.101,148.786
C09778=1125.535,-115.523,-45.623,179.585,4.096,148.785
C09779=1125.540,-115.739,-45.616,179.584,4.091,148.784
C09780=1125.544,-115.955,-45.609,179.585,4.087,148.783
C09781=1125.549,-116.171,-45.602,179.585,4.082,148.781
C09782=1125.554,-116.387,-45.595,179.585,4.078,148.780
C09783=1125.559,-116.603,-45.588,179.585,4.073,148.779
C09784=1125.564,-116.818,-45.580,179.585,4.068,148.778
C09785=1125.569,-117.068,-45.573,179.586,4.063,148.777
C09786=1125.574,-117.318,-45.565,179.586,4.057,148.776
C09787=1125.580,-117.568,-45.558,179.586,4.052,148.775
C09788=1125.585,-117.818,-45.549,179.586,4.046,148.773
C09789=1125.591,-118.067,-45.541,179.586,4.041,148.772
C09790=1125.596,-118.317,-45.533,179.586,4.036,148.771
C09791=1125.602,-118.567,-45.526,179.587,4.031,148.770
C09792=1125.607,-118.817,-45.517,179.587,4.026,148.769
C09793=1125.612,-119.067,-45.509,179.587,4.020,148.767
C09794=1125.618,-119.317,-45.501,179.587,4.014,148.766
C09795=1125.623,-119.566,-45.494,179.587,4.009,148.765
C09796=1125.629,-119.816,-45.485,179.587,4.004,148.764
C09797=1125.634,-120.066,-45.477,179.587,3.998,148.763
C09798=1125.640,-120.316,-45.470,179.587,3.993,148.761
C09799=1125.645,-120.566,-45.462,179.588,3.988,148.760
C09800=1125.651,-120.815,-45.455,179.587,3.982,148.759
C09801=1125.656,-121.066,-45.446,179.588,3.977,148.758
C09802=1125.661,-121.315,-45.439,179.588,3.971,148.757
C09803=1125.667,-121.565,-45.431,179.588,3.966,148.755
C09804=1125.672,-121.815,-45.423,179.588,3.960,148.754
C09805=1125.678,-122.064,-45.415,179.588,3.955,148.753
C09806=1125.683,-122.315,-45.407,179.589,3.950,148.752
C09807=1125.689,-122.564,-45.400,179.588,3.944,148.751
C09808=1125.695,-122.814,-45.392,179.589,3.939,148.749
C09809=1125.700,-123.064,-45.385,179.589,3.933,148.748
C09810=1125.705,-123.313,-45.376,179.589,3.927,148.747
C09811=1125.711,-123.563,-45.369,179.589,3.922,148.745
C09812=1125.716,-123.813,-45.361,179.590,3.917,148.744
C09813=1125.721,-124.063,-45.353,179.589,3.911,148.743
C09814=1125.727,-124.312,-45.346,179.590,3.906,148.742
C09815=1125.732,-124.563,-45.338,179.589,3.900,148.741
C09816=1125.738,-124.812,-45.331,179.590,3.894,148.739
C09817=1125.744,-125.062,-45.323,179.590,3.889,148.738
C09818=1125.748,-125.312,-45.315,179.590,3.883,148.737
C09819=1125.754,-125.562,-45.308,179.591,3.878,148.736
C09820=1125.760,-125.811,-45.300,179.590,3.872,148.734
C09821=1125.765,-126.062,-45.292,179.591,3.866,148.733
C09822=1125.771,-126.311,-45.285,179.591,3.861,148.732
C09823=1125.776,-126.561,-45.278,179.591,3.855,148.731
C09824=1125.781,-126.811,-45.269,179.591,3.850,148.730
C09825=1125.787,-127.061,-45.262,179.591,3.844,148.728
C09826=1125.793,-127.310,-45.254,179.591,3.839,148.727
C09827=1125.798,-127.561,-45.248,179.591,3.833,148.726
C09828=1125.803,-127.811,-45.240,179.591,3.827,148.724
C09829=1125.809,-128.060,-45.233,179.591,3.821,148.723
C09830=1125.815,-128.310,-45.225,179.592,3.816,148.722
C09831=1125.819,-128.560,-45.218,179.591,3.810,148.721
C09832=1125.825,-128.810,-45.210,179.592,3.805,148.719
C09833=1125.402,-128.800,-45.236,179.599,3.809,148.718
C09834=1125.396,-128.550,-45.243,179.599,3.814,148.719
C09835=1125.391,-128.301,-45.251,179.599,3.820,148.720
C09836=1125.386,-128.051,-45.258,179.598,3.826,148.722
C09837=1125.380,-127.801,-45.266,179.599,3.832,148.723
C09838=1125.375,-127.551,-45.273,179.598,3.837,148.724
C09839=1125.369,-127.301,-45.281,179.598,3.842,148.726
C09840=1125.364,-127.051,-45.289,179.598,3.848,148.727
C09841=1125.358,-126.802,-45.296,179.598,3.853,148.728
C09842=1125.353,-126.552,-45.304,179.598,3.860,148.729
C09843=1125.348,-126.302,-45.311,179.598,3.865,148.731
C09844=1125.342,-126.052,-45.319,179.598,3.871,148.732
C09845=1125.337,-125.802,-45.327,179.597,3.876,148.733
C09846=1125.331,-125.552,-45.334,179.597,3.881,148.734
C09847=1125.326,-125.303,-45.342,179.597,3.887,148.736
C09848=1125.320,-125.052,-45.350,179.597,3.893,148.737
C09849=1125.315,-124.803,-45.357,179.597,3.899,148.738
C09850=1125.309,-124.553,-45.365,179.597,3.904,148.739
C09851=1125.304,-124.303,-45.372,179.596,3.909,148.741
C09852=1125.298,-124.053,-45.380,179.597,3.915,148.742
C09853=1125.293,-123.804,-45.387,179.596,3.921,148.743
C09854=1125.287,-123.553,-45.396,179.596,3.926,148.744
C09855=1125.282,-123.304,-45.403,179.596,3.932,148.745
C09856=1125.276,-123.055,-45.411,179.596,3.937,148.747
C09857=1125.271,-122.805,-45.419,179.596,3.942,148.748
C09858=1125.265,-122.555,-45.427,179.596,3.948,148.749
C09859=1125.261,-122.305,-45.434,179.595,3.954,148.751
C09860=1125.255,-122.055,-45.442,179.595,3.959,148.752
C09861=1125.249,-121.805,-45.449,179.595,3.965,148.753
C09862=1125.244,-121.555,-45.458,179.595,3.970,148.754
C09863=1125.239,-121.306,-45.466,179.595,3.975,148.755
C09864=1125.233,-121.056,-45.474,179.595,3.981,148.757
C09865=1125.228,-120.806,-45.481,179.595,3.986,148.758
C09866=1125.222,-120.556,-45.489,179.594,3.992,148.759
C09867=1125.216,-120.306,-45.497,179.594,3.997,148.760
C09868=1125.211,-120.057,-45.505,179.594,4.003,148.761
C09869=1125.206,-119.807,-45.513,179.594,4.008,148.763
C09870=1125.200,-119.557,-45.520,179.594,4.013,148.764
C09871=1125.195,-119.307,-45.529,179.594,4.018,148.765
C09872=1125.189,-119.058,-45.537,179.594,4.024,148.766
C09873=1125.185,-118.807,-45.545,179.594,4.029,148.767
C09874=1125.178,-118.558,-45.552,179.593,4.035,148.769
C09875=1125.173,-118.307,-45.561,179.593,4.040,148.770
C09876=1125.168,-118.058,-45.569,179.593,4.046,148.771
C09877=1125.162,-117.808,-45.577,179.593,4.051,148.772
C09878=1125.157,-117.558,-45.584,179.593,4.056,148.773
C09879=1125.152,-117.309,-45.593,179.593,4.061,148.775
C09880=1125.146,-117.059,-45.601,179.592,4.066,148.776
C09881=1125.140,-116.808,-45.609,179.593,4.072,148.777
C09882=1125.136,-116.593,-45.615,179.592,4.077,148.778
C09883=1125.131,-116.377,-45.622,179.592,4.082,148.779
C09884=1125.126,-116.161,-45.629,179.592,4.086,148.780
C09885=1125.122,-115.946,-45.637,179.591,4.091,148.781
C09886=1125.117,-115.730,-45.643,179.592,4.096,148.782
C09887=1125.113,-115.514,-45.651,179.591,4.100,148.783
C09888=1125.108,-115.298,-45.657,179.591,4.105,148.784
C09889=1125.102,-115.082,-45.664,179.591,4.109,148.785
C09890=1125.098,-114.833,-45.673,179.591,4.115,148.787
C09891=1125.092,-114.583,-45.680,179.591,4.120,148.788
C09892=1125.086,-114.333,-45.689,179.590,4.125,148.789
C09893=1125.081,-114.083,-45.697,179.590,4.130,148.790
C09894=1125.076,-113.833,-45.705,179.590,4.135,148.791
C09895=1125.071,-113.583,-45.714,179.590,4.141,148.793
C09896=1125.065,-113.334,-45.721,179.589,4.146,148.794
C09897=1125.060,-113.084,-45.730,179.589,4.151,148.795
C09898=1125.053,-112.834,-45.738,179.589,4.156,148.796
C09899=1125.049,-112.584,-45.746,179.589,4.162,148.797
C09900=1125.043,-112.335,-45.754,179.589,4.167,148.798
C09901=1125.038,-112.084,-45.762,179.589,4.172,148.800
C09902=1125.032,-111.834,-45.771,179.589,4.177,148.801
C09903=1125.027,-111.585,-45.779,179.589,4.182,148.802
C09904=1125.022,-111.335,-45.787,179.588,4.188,148.803
C09905=1125.016,-111.086,-45.796,179.588,4.193,148.804
C09906=1125.011,-110.836,-45.804,179.588,4.198,148.806
C09907=1125.005,-110.586,-45.813,179.588,4.203,148.807
C09908=1124.999,-110.336,-45.821,179.587,4.208,148.808
C09909=1124.995,-110.086,-45.829,179.587,4.213,148.809
C09910=1124.989,-109.837,-45.837,179.587,4.219,148.810
C09911=1124.984,-109.587,-45.846,179.587,4.224,148.812
C09912=1124.978,-109.336,-45.854,179.586,4.229,148.813
C09913=1124.972,-109.087,-45.863,179.586,4.234,148.814
C09914=1124.967,-108.837,-45.872,179.586,4.239,148.815
C09915=1124.962,-108.587,-45.880,179.586,4.244,148.816
C09916=1124.957,-108.338,-45.888,179.586,4.249,148.817
C09917=1124.951,-108.087,-45.896,179.586,4.254,148.818
C09918=1124.946,-107.838,-45.904,179.585,4.260,148.820
C09919=1124.940,-107.588,-45.913,179.585,4.265,148.821
C09920=1124.935,-107.338,-45.921,179.585,4.270,148.822
C09921=1124.929,-107.089,-45.930,179.585,4.275,148.823
C09922=1124.924,-106.839,-45.939,179.584,4.280,148.824
C09923=1124.919,-106.589,-45.947,179.584,4.285,148.826
C09924=1124.913,-106.339,-45.956,179.584,4.291,148.827
C09925=1124.908,-106.090,-45.964,179.584,4.296,148.828
C09926=1124.902,-105.839,-45.973,179.584,4.301,148.829
C09927=1124.898,-105.590,-45.981,179.584,4.306,148.830
C09928=1124.892,-105.340,-45.990,179.584,4.311,148.831
C09929=1124.887,-105.091,-45.998,179.583,4.316,148.833
C09930=1124.881,-104.840,-46.007,179.583,4.321,148.834
C09931=1124.875,-104.591,-46.015,179.583,4.326,148.835
C09932=1124.870,-104.341,-46.024,179.583,4.332,148.836
C09933=1124.865,-104.091,-46.033,179.582,4.337,148.837
C09934=1124.860,-103.841,-46.041,179.582,4.341,148.839
C09935=1124.854,-103.592,-46.050,179.581,4.346,148.840
C09936=1124.849,-103.342,-46.059,179.581,4.351,148.841
C09937=1124.844,-103.092,-46.067,179.581,4.357,148.842
C09938=1124.838,-102.876,-46.074,179.581,4.361,148.843
C09939=1124.834,-102.660,-46.082,179.581,4.365,148.844
C09940=1124.829,-102.445,-46.089,179.581,4.369,148.845
C09941=1124.825,-102.229,-46.097,179.581,4.374,148.846
C09942=1124.820,-102.013,-46.104,179.580,4.379,148.847
C09943=1124.816,-101.797,-46.112,179.580,4.383,148.848
C09944=1124.811,-101.582,-46.120,179.580,4.387,148.849
C09945=1124.806,-101.366,-46.127,179.580,4.391,148.850
C09946=1124.801,-101.116,-46.136,179.579,4.396,148.851
C09947=1124.795,-100.867,-46.144,179.579,4.402,148.852
C09948=1124.790,-100.617,-46.153,179.579,4.407,148.854
C09949=1124.784,-100.367,-46.163,179.578,4.411,148.855
C09950=1124.779,-100.117,-46.172,179.578,4.416,148.856
C09951=1124.773,-99.867,-46.179,179.578,4.421,148.857
C09952=1124.768,-99.617,-46.188,179.578,4.427,148.858
C09953=1124.763,-99.367,-46.197,179.577,4.432,148.859
C09954=1124.758,-99.118,-46.206,179.577,4.437,148.861
C09955=1124.752,-98.868,-46.215,179.577,4.441,148.862
C09956=1124.747,-98.619,-46.224,179.577,4.446,148.863
C09957=1124.741,-98.369,-46.232,179.576,4.451,148.864
C09958=1124.736,-98.119,-46.241,179.576,4.456,148.865
C09959=1124.730,-97.869,-46.251,179.576,4.462,148.866
C09960=1124.725,-97.619,-46.260,179.576,4.467,148.868
C09961=1124.719,-97.370,-46.268,179.575,4.471,148.869
C09962=1124.714,-97.120,-46.277,179.575,4.476,148.870
C09963=1124.709,-96.870,-46.286,179.575,4.481,148.871
C09964=1124.704,-96.620,-46.295,179.574,4.487,148.872
C09965=1124.699,-96.370,-46.304,179.574,4.491,148.873
C09966=1124.692,-96.121,-46.313,179.574,4.496,148.874
C09967=1124.687,-95.871,-46.322,179.574,4.501,148.876
C09968=1124.682,-95.621,-46.331,179.573,4.506,148.877
C09969=1124.677,-95.371,-46.340,179.573,4.511,148.878
C09970=1124.672,-95.121,-46.349,179.572,4.516,148.879
C09971=1124.666,-94.872,-46.358,179.572,4.521,148.880
C09972=1124.660,-94.621,-46.367,179.572,4.526,148.881
C09973=1124.655,-94.372,-46.376,179.571,4.530,148.883
C09974=1124.650,-94.122,-46.384,179.571,4.536,148.884
C09975=1124.644,-93.873,-46.393,179.570,4.540,148.885
C09976=1124.639,-93.623,-46.402,179.569,4.545,148.886
C09977=1124.633,-93.373,-46.412,179.569,4.550,148.888
C09978=1124.628,-93.123,-46.421,179.568,4.554,148.889
C09979=1124.623,-92.873,-46.430,179.567,4.559,148.890
C09980=1124.618,-92.623,-46.438,179.566,4.564,148.891
C09981=1124.612,-92.374,-46.448,179.566,4.568,148.893
C09982=1124.606,-92.124,-46.457,179.565,4.573,148.894
C09983=1124.601,-91.874,-46.466,179.564,4.578,148.895
C09984=1124.596,-91.625,-46.475,179.563,4.583,148.896
C09985=1124.590,-91.374,-46.484,179.563,4.588,148.898
C09986=1124.585,-91.125,-46.493,179.562,4.592,148.899
C09987=1124.580,-90.875,-46.502,179.562,4.597,148.900
C09988=1124.575,-90.625,-46.511,179.561,4.602,148.901
C09989=1124.569,-90.375,-46.521,179.560,4.606,148.903
C09990=1124.564,-90.126,-46.530,179.560,4.612,148.904
C09991=1124.558,-89.876,-46.539,179.559,4.616,148.905
C09992=1124.553,-89.627,-46.548,179.558,4.622,148.906
C09993=1124.547,-89.376,-46.557,179.558,4.626,148.908
C09994=1124.543,-89.161,-46.565,179.558,4.631,148.908
C09995=1124.539,-88.945,-46.573,179.557,4.635,148.910
C09996=1124.534,-88.730,-46.581,179.557,4.639,148.911
//INST
///DATE 2021/06/25 14:33
///ATTR SC,RW,RJ
////FRAME ROBOT
///GROUP1 RB1
NOP
MOVL C00000 V=800.0 PL=0
MOVL C00001 V=800.0 PL=0
MOVL C00002 V=800.0 PL=0
MOVL C00003 V=800.0 PL=0
MOVL C00004 V=800.0 PL=0
MOVL C00005 V=800.0 PL=0
MOVL C00006 V=800.0 PL=0
MOVL C00007 V=800.0 PL=0
MOVL C00008 V=800.0 PL=0
MOVL C00009 V=800.0 PL=0
MOVL C00010 V=800.0 PL=0
MOVL C00011 V=800.0 PL=0
MOVL C00012 V=800.0 PL=0
MOVL C00013 V=800.0 PL=0
MOVL C00014 V=800.0 PL=0
MOVL C00015 V=800.0 PL=0
MOVL C00016 V=800.0 PL=0
MOVL C00017 V=800.0 PL=0
MOVL C00018 V=800.0 PL=0
MOVL C00019 V=800.0 PL=0
MOVL C00020 V=800.0 PL=0
MOVL C00021 V=800.0 PL=0
MOVL C00022 V=800.0 PL=0
MOVL C00023 V=800.0 PL=0
MOVL C00024 V=800.0 PL=0
MOVL C00025 V=800.0 PL=0
MOVL C00026 V=800.0 PL=0
MOVL C00027 V=800.0 PL=0
MOVL C00028 V=800.0 PL=0
MOVL C00029 V=800.0 PL=0
MOVL C00030 V=800.0 PL=0
MOVL C00031 V=800.0 PL=0
MOVL C00032 V=800.0 PL=0
MOVL C00033 V=800.0 PL=0
MOVL C00034 V=800.0 PL=0
MOVL C00035 V=800.0 PL=0
MOVL C00036 V=800.0 PL=0
MOVL C00037 V=800.0 PL=0
MOVL C00038 V=800.0 PL=0
MOVL C00039 V=800.0 PL=0
MOVL C00040 V=800.0 PL=0
MOVL C00041 V=800.0 PL=0
MOVL C00042 V=800.0 PL=0
MOVL C00043 V=800.0 PL=0
MOVL C00044 V=800.0 PL=0
MOVL C00045 V=800.0 PL=0
MOVL C00046 V=800.0 PL=0
MOVL C00047 V=800.0 PL=0
MOVL C00048 V=800.0 PL=0
MOVL C00049 V=800.0 PL=0
MOVL C00050 V=800.0 PL=0
MOVL C00051 V=800.0 PL=0
MOVL C00052 V=800.0 PL=0
MOVL C00053 V=800.0 PL=0
MOVL C00054 V=800.0 PL=0
MOVL C00055 V=800.0 PL=0
MOVL C00056 V=800.0 PL=0
MOVL C00057 V=800.0 PL=0
MOVL C00058 V=800.0 PL=0
MOVL C00059 V=800.0 PL=0
MOVL C00060 V=800.0 PL=0
MOVL C00061 V=800.0 PL=0
MOVL C00062 V=800.0 PL=0
MOVL C00063 V=800.0 PL=0
MOVL C00064 V=800.0 PL=0
MOVL C00065 V=800.0 PL=0
MOVL C00066 V=800.0 PL=0
MOVL C00067 V=800.0 PL=0
MOVL C00068 V=800.0 PL=0
MOVL C00069 V=800.0 PL=0
MOVL C00070 V=800.0 PL=0
MOVL C00071 V=800.0 PL=0
MOVL C00072 V=800.0 PL=0
MOVL C00073 V=800.0 PL=0
MOVL C00074 V=800.0 PL=0
MOVL C00075 V=800.0 PL=0
MOVL C00076 V=800.0 PL=0
MOVL C00077 V=800.0 PL=0
MOVL C00078 V=800.0 PL=0
MOVL C00079 V=800.0 PL=0
MOVL C00080 V=800.0 PL=0
MOVL C00081 V=800.0 PL=0
MOVL C00082 V=800.0 PL=0
MOVL C00083 V=800.0 PL=0
MOVL C00084 V=800.0 PL=0
MOVL C00085 V=800.0 PL=0
MOVL C00086 V=800.0 PL=0
MOVL C00087 V=800.0 PL=0
MOVL C00088 V=800.0 PL=0
MOVL C00089 V=800.0 PL=0
MOVL C00090 V=800.0 PL=0
MOVL C00091 V=800.0 PL=0
MOVL C00092 V=800.0 PL=0
MOVL C00093 V=800.0 PL=0
MOVL C00094 V=800.0 PL=0
MOVL C00095 V=800.0 PL=0
MOVL C00096 V=800.0 PL=0
MOVL C00097 V=800.0 PL=0
MOVL C00098 V=800.0 PL=0
MOVL C00099 V=800.0 PL=0
MOVL C00100 V=800.0 PL=0
MOVL C00101 V=800.0 PL=0
MOVL C00102 V=800.0 PL=0
MOVL C00103 V=800.0 PL=0
MOVL C00104 V=800.0 PL=0
MOVL C00105 V=800.0 PL=0
MOVL C00106 V=800.0 PL=0
MOVL C00107 V=800.0 PL=0
MOVL C00108 V=800.0 PL=0
MOVL C00109 V=800.0 PL=0
MOVL C00110 V=800.0 PL=0
MOVL C00111 V=800.0 PL=0
MOVL C00112 V=800.0 PL=0
MOVL C00113 V=800.0 PL=0
MOVL C00114 V=800.0 PL=0
MOVL C00115 V=800.0 PL=0
MOVL C00116 V=800.0 PL=0
MOVL C00117 V=800.0 PL=0
MOVL C00118 V=800.0 PL=0
MOVL C00119 V=800.0 PL=0
MOVL C00120 V=800.0 PL=0
MOVL C00121 V=800.0 PL=0
MOVL C00122 V=800.0 PL=0
MOVL C00123 V=800.0 PL=0
MOVL C00124 V=800.0 PL=0
MOVL C00125 V=800.0 PL=0
MOVL C00126 V=800.0 PL=0
MOVL C00127 V=800.0 PL=0
MOVL C00128 V=800.0 PL=0
MOVL C00129 V=800.0 PL=0
MOVL C00130 V=800.0 PL=0
MOVL C00131 V=800.0 PL=0
MOVL C00132 V=800.0 PL=0
MOVL C00133 V=800.0 PL=0
MOVL C00134 V=800.0 PL=0
MOVL C00135 V=800.0 PL=0
MOVL C00136 V=800.0 PL=0
MOVL C00137 V=800.0 PL=0
MOVL C00138 V=800.0 PL=0
MOVL C00139 V=800.0 PL=0
MOVL C00140 V=800.0 PL=0
MOVL C00141 V=800.0 PL=0
MOVL C00142 V=800.0 PL=0
MOVL C00143 V=800.0 PL=0
MOVL C00144 V=800.0 PL=0
MOVL C00145 V=800.0 PL=0
MOVL C00146 V=800.0 PL=0
MOVL C00147 V=800.0 PL=0
MOVL C00148 V=800.0 PL=0
MOVL C00149 V=800.0 PL=0
MOVL C00150 V=800.0 PL=0
MOVL C00151 V=800.0 PL=0
MOVL C00152 V=800.0 PL=0
MOVL C00153 V=800.0 PL=0
MOVL C00154 V=800.0 PL=0
MOVL C00155 V=800.0 PL=0
MOVL C00156 V=800.0 PL=0
MOVL C00157 V=800.0 PL=0
MOVL C00158 V=800.0 PL=0
MOVL C00159 V=800.0 PL=0
MOVL C00160 V=800.0 PL=0
MOVL C00161 V=800.0 PL=0
MOVL C00162 V=800.0 PL=0
MOVL C00163 V=800.0 PL=0
MOVL C00164 V=800.0 PL=0
MOVL C00165 V=800.0 PL=0
MOVL C00166 V=800.0 PL=0
MOVL C00167 V=800.0 PL=0
MOVL C00168 V=800.0 PL=0
MOVL C00169 V=800.0 PL=0
MOVL C00170 V=800.0 PL=0
MOVL C00171 V=800.0 PL=0
MOVL C00172 V=800.0 PL=0
MOVL C00173 V=800.0 PL=0
MOVL C00174 V=800.0 PL=0
MOVL C00175 V=800.0 PL=0
MOVL C00176 V=800.0 PL=0
MOVL C00177 V=800.0 PL=0
MOVL C00178 V=800.0 PL=0
MOVL C00179 V=800.0 PL=0
MOVL C00180 V=800.0 PL=0
MOVL C00181 V=800.0 PL=0
MOVL C00182 V=800.0 PL=0
MOVL C00183 V=800.0 PL=0
MOVL C00184 V=800.0 PL=0
MOVL C00185 V=800.0 PL=0
MOVL C00186 V=800.0 PL=0
MOVL C00187 V=800.0 PL=0
MOVL C00188 V=800.0 PL=0
MOVL C00189 V=800.0 PL=0
MOVL C00190 V=800.0 PL=0
MOVL C00191 V=800.0 PL=0
MOVL C00192 V=800.0 PL=0
MOVL C00193 V=800.0 PL=0
MOVL C00194 V=800.0 PL=0
MOVL C00195 V=800.0 PL=0
MOVL C00196 V=800.0 PL=0
MOVL C00197 V=800.0 PL=0
MOVL C00198 V=800.0 PL=0
MOVL C00199 V=800.0 PL=0
MOVL C00200 V=800.0 PL=0
MOVL C00201 V=800.0 PL=0
MOVL C00202 V=800.0 PL=0
MOVL C00203 V=800.0 PL=0
MOVL C00204 V=800.0 PL=0
MOVL C00205 V=800.0 PL=0
MOVL C00206 V=800.0 PL=0
MOVL C00207 V=800.0 PL=0
MOVL C00208 V=800.0 PL=0
MOVL C00209 V=800.0 PL=0
MOVL C00210 V=800.0 PL=0
MOVL C00211 V=800.0 PL=0
MOVL C00212 V=800.0 PL=0
MOVL C00213 V=800.0 PL=0
MOVL C00214 V=800.0 PL=0
MOVL C00215 V=800.0 PL=0
MOVL C00216 V=800.0 PL=0
MOVL C00217 V=800.0 PL=0
MOVL C00218 V=800.0 PL=0
MOVL C00219 V=800.0 PL=0
MOVL C00220 V=800.0 PL=0
MOVL C00221 V=800.0 PL=0
MOVL C00222 V=800.0 PL=0
MOVL C00223 V=800.0 PL=0
MOVL C00224 V=800.0 PL=0
MOVL C00225 V=800.0 PL=0
MOVL C00226 V=800.0 PL=0
MOVL C00227 V=800.0 PL=0
MOVL C00228 V=800.0 PL=0
MOVL C00229 V=800.0 PL=0
MOVL C00230 V=800.0 PL=0
MOVL C00231 V=800.0 PL=0
MOVL C00232 V=800.0 PL=0
MOVL C00233 V=800.0 PL=0
MOVL C00234 V=800.0 PL=0
MOVL C00235 V=800.0 PL=0
MOVL C00236 V=800.0 PL=0
MOVL C00237 V=800.0 PL=0
MOVL C00238 V=800.0 PL=0
MOVL C00239 V=800.0 PL=0
MOVL C00240 V=800.0 PL=0
MOVL C00241 V=800.0 PL=0
MOVL C00242 V=800.0 PL=0
MOVL C00243 V=800.0 PL=0
MOVL C00244 V=800.0 PL=0
MOVL C00245 V=800.0 PL=0
MOVL C00246 V=800.0 PL=0
MOVL C00247 V=800.0 PL=0
MOVL C00248 V=800.0 PL=0
MOVL C00249 V=800.0 PL=0
MOVL C00250 V=800.0 PL=0
MOVL C00251 V=800.0 PL=0
MOVL C00252 V=800.0 PL=0
MOVL C00253 V=800.0 PL=0
MOVL C00254 V=800.0 PL=0
MOVL C00255 V=800.0 PL=0
MOVL C00256 V=800.0 PL=0
MOVL C00257 V=800.0 PL=0
MOVL C00258 V=800.0 PL=0
MOVL C00259 V=800.0 PL=0
MOVL C00260 V=800.0 PL=0
MOVL C00261 V=800.0 PL=0
MOVL C00262 V=800.0 PL=0
MOVL C00263 V=800.0 PL=0
MOVL C00264 V=800.0 PL=0
MOVL C00265 V=800.0 PL=0
MOVL C00266 V=800.0 PL=0
MOVL C00267 V=800.0 PL=0
MOVL C00268 V=800.0 PL=0
MOVL C00269 V=800.0 PL=0
MOVL C00270 V=800.0 PL=0
MOVL C00271 V=800.0 PL=0
MOVL C00272 V=800.0 PL=0
MOVL C00273 V=800.0 PL=0
MOVL C00274 V=800.0 PL=0
MOVL C00275 V=800.0 PL=0
MOVL C00276 V=800.0 PL=0
MOVL C00277 V=800.0 PL=0
MOVL C00278 V=800.0 PL=0
MOVL C00279 V=800.0 PL=0
MOVL C00280 V=800.0 PL=0
MOVL C00281 V=800.0 PL=0
MOVL C00282 V=800.0 PL=0
MOVL C00283 V=800.0 PL=0
MOVL C00284 V=800.0 PL=0
MOVL C00285 V=800.0 PL=0
MOVL C00286 V=800.0 PL=0
MOVL C00287 V=800.0 PL=0
MOVL C00288 V=800.0 PL=0
MOVL C00289 V=800.0 PL=0
MOVL C00290 V=800.0 PL=0
MOVL C00291 V=800.0 PL=0
MOVL C00292 V=800.0 PL=0
MOVL C00293 V=800.0 PL=0
MOVL C00294 V=800.0 PL=0
MOVL C00295 V=800.0 PL=0
MOVL C00296 V=800.0 PL=0
MOVL C00297 V=800.0 PL=0
MOVL C00298 V=800.0 PL=0
MOVL C00299 V=800.0 PL=0
MOVL C00300 V=800.0 PL=0
MOVL C00301 V=800.0 PL=0
MOVL C00302 V=800.0 PL=0
MOVL C00303 V=800.0 PL=0
MOVL C00304 V=800.0 PL=0
MOVL C00305 V=800.0 PL=0
MOVL C00306 V=800.0 PL=0
MOVL C00307 V=800.0 PL=0
MOVL C00308 V=800.0 PL=0
MOVL C00309 V=800.0 PL=0
MOVL C00310 V=800.0 PL=0
MOVL C00311 V=800.0 PL=0
MOVL C00312 V=800.0 PL=0
MOVL C00313 V=800.0 PL=0
MOVL C00314 V=800.0 PL=0
MOVL C00315 V=800.0 PL=0
MOVL C00316 V=800.0 PL=0
MOVL C00317 V=800.0 PL=0
MOVL C00318 V=800.0 PL=0
MOVL C00319 V=800.0 PL=0
MOVL C00320 V=800.0 PL=0
MOVL C00321 V=800.0 PL=0
MOVL C00322 V=800.0 PL=0
MOVL C00323 V=800.0 PL=0
MOVL C00324 V=800.0 PL=0
MOVL C00325 V=800.0 PL=0
MOVL C00326 V=800.0 PL=0
MOVL C00327 V=800.0 PL=0
MOVL C00328 V=800.0 PL=0
MOVL C00329 V=800.0 PL=0
MOVL C00330 V=800.0 PL=0
MOVL C00331 V=800.0 PL=0
MOVL C00332 V=800.0 PL=0
MOVL C00333 V=800.0 PL=0
MOVL C00334 V=800.0 PL=0
MOVL C00335 V=800.0 PL=0
MOVL C00336 V=800.0 PL=0
MOVL C00337 V=800.0 PL=0
MOVL C00338 V=800.0 PL=0
MOVL C00339 V=800.0 PL=0
MOVL C00340 V=800.0 PL=0
MOVL C00341 V=800.0 PL=0
MOVL C00342 V=800.0 PL=0
MOVL C00343 V=800.0 PL=0
MOVL C00344 V=800.0 PL=0
MOVL C00345 V=800.0 PL=0
MOVL C00346 V=800.0 PL=0
MOVL C00347 V=800.0 PL=0
MOVL C00348 V=800.0 PL=0
MOVL C00349 V=800.0 PL=0
MOVL C00350 V=800.0 PL=0
MOVL C00351 V=800.0 PL=0
MOVL C00352 V=800.0 PL=0
MOVL C00353 V=800.0 PL=0
MOVL C00354 V=800.0 PL=0
MOVL C00355 V=800.0 PL=0
MOVL C00356 V=800.0 PL=0
MOVL C00357 V=800.0 PL=0
MOVL C00358 V=800.0 PL=0
MOVL C00359 V=800.0 PL=0
MOVL C00360 V=800.0 PL=0
MOVL C00361 V=800.0 PL=0
MOVL C00362 V=800.0 PL=0
MOVL C00363 V=800.0 PL=0
MOVL C00364 V=800.0 PL=0
MOVL C00365 V=800.0 PL=0
MOVL C00366 V=800.0 PL=0
MOVL C00367 V=800.0 PL=0
MOVL C00368 V=800.0 PL=0
MOVL C00369 V=800.0 PL=0
MOVL C00370 V=800.0 PL=0
MOVL C00371 V=800.0 PL=0
MOVL C00372 V=800.0 PL=0
MOVL C00373 V=800.0 PL=0
MOVL C00374 V=800.0 PL=0
MOVL C00375 V=800.0 PL=0
MOVL C00376 V=800.0 PL=0
MOVL C00377 V=800.0 PL=0
MOVL C00378 V=800.0 PL=0
MOVL C00379 V=800.0 PL=0
MOVL C00380 V=800.0 PL=0
MOVL C00381 V=800.0 PL=0
MOVL C00382 V=800.0 PL=0
MOVL C00383 V=800.0 PL=0
MOVL C00384 V=800.0 PL=0
MOVL C00385 V=800.0 PL=0
MOVL C00386 V=800.0 PL=0
MOVL C00387 V=800.0 PL=0
MOVL C00388 V=800.0 PL=0
MOVL C00389 V=800.0 PL=0
MOVL C00390 V=800.0 PL=0
MOVL C00391 V=800.0 PL=0
MOVL C00392 V=800.0 PL=0
MOVL C00393 V=800.0 PL=0
MOVL C00394 V=800.0 PL=0
MOVL C00395 V=800.0 PL=0
MOVL C00396 V=800.0 PL=0
MOVL C00397 V=800.0 PL=0
MOVL C00398 V=800.0 PL=0
MOVL C00399 V=800.0 PL=0
MOVL C00400 V=800.0 PL=0
MOVL C00401 V=800.0 PL=0
MOVL C00402 V=800.0 PL=0
MOVL C00403 V=800.0 PL=0
MOVL C00404 V=800.0 PL=0
MOVL C00405 V=800.0 PL=0
MOVL C00406 V=800.0 PL=0
MOVL C00407 V=800.0 PL=0
MOVL C00408 V=800.0 PL=0
MOVL C00409 V=800.0 PL=0
MOVL C00410 V=800.0 PL=0
MOVL C00411 V=800.0 PL=0
MOVL C00412 V=800.0 PL=0
MOVL C00413 V=800.0 PL=0
MOVL C00414 V=800.0 PL=0
MOVL C00415 V=800.0 PL=0
MOVL C00416 V=800.0 PL=0
MOVL C00417 V=800.0 PL=0
MOVL C00418 V=800.0 PL=0
MOVL C00419 V=800.0 PL=0
MOVL C00420 V=800.0 PL=0
MOVL C00421 V=800.0 PL=0
MOVL C00422 V=800.0 PL=0
MOVL C00423 V=800.0 PL=0
MOVL C00424 V=800.0 PL=0
MOVL C00425 V=800.0 PL=0
MOVL C00426 V=800.0 PL=0
MOVL C00427 V=800.0 PL=0
MOVL C00428 V=800.0 PL=0
MOVL C00429 V=800.0 PL=0
MOVL C00430 V=800.0 PL=0
MOVL C00431 V=800.0 PL=0
MOVL C00432 V=800.0 PL=0
MOVL C00433 V=800.0 PL=0
MOVL C00434 V=800.0 PL=0
MOVL C00435 V=800.0 PL=0
MOVL C00436 V=800.0 PL=0
MOVL C00437 V=800.0 PL=0
MOVL C00438 V=800.0 PL=0
MOVL C00439 V=800.0 PL=0
MOVL C00440 V=800.0 PL=0
MOVL C00441 V=800.0 PL=0
MOVL C00442 V=800.0 PL=0
MOVL C00443 V=800.0 PL=0
MOVL C00444 V=800.0 PL=0
MOVL C00445 V=800.0 PL=0
MOVL C00446 V=800.0 PL=0
MOVL C00447 V=800.0 PL=0
MOVL C00448 V=800.0 PL=0
MOVL C00449 V=800.0 PL=0
MOVL C00450 V=800.0 PL=0
MOVL C00451 V=800.0 PL=0
MOVL C00452 V=800.0 PL=0
MOVL C00453 V=800.0 PL=0
MOVL C00454 V=800.0 PL=0
MOVL C00455 V=800.0 PL=0
MOVL C00456 V=800.0 PL=0
MOVL C00457 V=800.0 PL=0
MOVL C00458 V=800.0 PL=0
MOVL C00459 V=800.0 PL=0
MOVL C00460 V=800.0 PL=0
MOVL C00461 V=800.0 PL=0
MOVL C00462 V=800.0 PL=0
MOVL C00463 V=800.0 PL=0
MOVL C00464 V=800.0 PL=0
MOVL C00465 V=800.0 PL=0
MOVL C00466 V=800.0 PL=0
MOVL C00467 V=800.0 PL=0
MOVL C00468 V=800.0 PL=0
MOVL C00469 V=800.0 PL=0
MOVL C00470 V=800.0 PL=0
MOVL C00471 V=800.0 PL=0
MOVL C00472 V=800.0 PL=0
MOVL C00473 V=800.0 PL=0
MOVL C00474 V=800.0 PL=0
MOVL C00475 V=800.0 PL=0
MOVL C00476 V=800.0 PL=0
MOVL C00477 V=800.0 PL=0
MOVL C00478 V=800.0 PL=0
MOVL C00479 V=800.0 PL=0
MOVL C00480 V=800.0 PL=0
MOVL C00481 V=800.0 PL=0
MOVL C00482 V=800.0 PL=0
MOVL C00483 V=800.0 PL=0
MOVL C00484 V=800.0 PL=0
MOVL C00485 V=800.0 PL=0
MOVL C00486 V=800.0 PL=0
MOVL C00487 V=800.0 PL=0
MOVL C00488 V=800.0 PL=0
MOVL C00489 V=800.0 PL=0
MOVL C00490 V=800.0 PL=0
MOVL C00491 V=800.0 PL=0
MOVL C00492 V=800.0 PL=0
MOVL C00493 V=800.0 PL=0
MOVL C00494 V=800.0 PL=0
MOVL C00495 V=800.0 PL=0
MOVL C00496 V=800.0 PL=0
MOVL C00497 V=800.0 PL=0
MOVL C00498 V=800.0 PL=0
MOVL C00499 V=800.0 PL=0
MOVL C00500 V=800.0 PL=0
MOVL C00501 V=800.0 PL=0
MOVL C00502 V=800.0 PL=0
MOVL C00503 V=800.0 PL=0
MOVL C00504 V=800.0 PL=0
MOVL C00505 V=800.0 PL=0
MOVL C00506 V=800.0 PL=0
MOVL C00507 V=800.0 PL=0
MOVL C00508 V=800.0 PL=0
MOVL C00509 V=800.0 PL=0
MOVL C00510 V=800.0 PL=0
MOVL C00511 V=800.0 PL=0
MOVL C00512 V=800.0 PL=0
MOVL C00513 V=800.0 PL=0
MOVL C00514 V=800.0 PL=0
MOVL C00515 V=800.0 PL=0
MOVL C00516 V=800.0 PL=0
MOVL C00517 V=800.0 PL=0
MOVL C00518 V=800.0 PL=0
MOVL C00519 V=800.0 PL=0
MOVL C00520 V=800.0 PL=0
MOVL C00521 V=800.0 PL=0
MOVL C00522 V=800.0 PL=0
MOVL C00523 V=800.0 PL=0
MOVL C00524 V=800.0 PL=0
MOVL C00525 V=800.0 PL=0
MOVL C00526 V=800.0 PL=0
MOVL C00527 V=800.0 PL=0
MOVL C00528 V=800.0 PL=0
MOVL C00529 V=800.0 PL=0
MOVL C00530 V=800.0 PL=0
MOVL C00531 V=800.0 PL=0
MOVL C00532 V=800.0 PL=0
MOVL C00533 V=800.0 PL=0
MOVL C00534 V=800.0 PL=0
MOVL C00535 V=800.0 PL=0
MOVL C00536 V=800.0 PL=0
MOVL C00537 V=800.0 PL=0
MOVL C00538 V=800.0 PL=0
MOVL C00539 V=800.0 PL=0
MOVL C00540 V=800.0 PL=0
MOVL C00541 V=800.0 PL=0
MOVL C00542 V=800.0 PL=0
MOVL C00543 V=800.0 PL=0
MOVL C00544 V=800.0 PL=0
MOVL C00545 V=800.0 PL=0
MOVL C00546 V=800.0 PL=0
MOVL C00547 V=800.0 PL=0
MOVL C00548 V=800.0 PL=0
MOVL C00549 V=800.0 PL=0
MOVL C00550 V=800.0 PL=0
MOVL C00551 V=800.0 PL=0
MOVL C00552 V=800.0 PL=0
MOVL C00553 V=800.0 PL=0
MOVL C00554 V=800.0 PL=0
MOVL C00555 V=800.0 PL=0
MOVL C00556 V=800.0 PL=0
MOVL C00557 V=800.0 PL=0
MOVL C00558 V=800.0 PL=0
MOVL C00559 V=800.0 PL=0
MOVL C00560 V=800.0 PL=0
MOVL C00561 V=800.0 PL=0
MOVL C00562 V=800.0 PL=0
MOVL C00563 V=800.0 PL=0
MOVL C00564 V=800.0 PL=0
MOVL C00565 V=800.0 PL=0
MOVL C00566 V=800.0 PL=0
MOVL C00567 V=800.0 PL=0
MOVL C00568 V=800.0 PL=0
MOVL C00569 V=800.0 PL=0
MOVL C00570 V=800.0 PL=0
MOVL C00571 V=800.0 PL=0
MOVL C00572 V=800.0 PL=0
MOVL C00573 V=800.0 PL=0
MOVL C00574 V=800.0 PL=0
MOVL C00575 V=800.0 PL=0
MOVL C00576 V=800.0 PL=0
MOVL C00577 V=800.0 PL=0
MOVL C00578 V=800.0 PL=0
MOVL C00579 V=800.0 PL=0
MOVL C00580 V=800.0 PL=0
MOVL C00581 V=800.0 PL=0
MOVL C00582 V=800.0 PL=0
MOVL C00583 V=800.0 PL=0
MOVL C00584 V=800.0 PL=0
MOVL C00585 V=800.0 PL=0
MOVL C00586 V=800.0 PL=0
MOVL C00587 V=800.0 PL=0
MOVL C00588 V=800.0 PL=0
MOVL C00589 V=800.0 PL=0
MOVL C00590 V=800.0 PL=0
MOVL C00591 V=800.0 PL=0
MOVL C00592 V=800.0 PL=0
MOVL C00593 V=800.0 PL=0
MOVL C00594 V=800.0 PL=0
MOVL C00595 V=800.0 PL=0
MOVL C00596 V=800.0 PL=0
MOVL C00597 V=800.0 PL=0
MOVL C00598 V=800.0 PL=0
MOVL C00599 V=800.0 PL=0
MOVL C00600 V=800.0 PL=0
MOVL C00601 V=800.0 PL=0
MOVL C00602 V=800.0 PL=0
MOVL C00603 V=800.0 PL=0
MOVL C00604 V=800.0 PL=0
MOVL C00605 V=800.0 PL=0
MOVL C00606 V=800.0 PL=0
MOVL C00607 V=800.0 PL=0
MOVL C00608 V=800.0 PL=0
MOVL C00609 V=800.0 PL=0
MOVL C00610 V=800.0 PL=0
MOVL C00611 V=800.0 PL=0
MOVL C00612 V=800.0 PL=0
MOVL C00613 V=800.0 PL=0
MOVL C00614 V=800.0 PL=0
MOVL C00615 V=800.0 PL=0
MOVL C00616 V=800.0 PL=0
MOVL C00617 V=800.0 PL=0
MOVL C00618 V=800.0 PL=0
MOVL C00619 V=800.0 PL=0
MOVL C00620 V=800.0 PL=0
MOVL C00621 V=800.0 PL=0
MOVL C00622 V=800.0 PL=0
MOVL C00623 V=800.0 PL=0
MOVL C00624 V=800.0 PL=0
MOVL C00625 V=800.0 PL=0
MOVL C00626 V=800.0 PL=0
MOVL C00627 V=800.0 PL=0
MOVL C00628 V=800.0 PL=0
MOVL C00629 V=800.0 PL=0
MOVL C00630 V=800.0 PL=0
MOVL C00631 V=800.0 PL=0
MOVL C00632 V=800.0 PL=0
MOVL C00633 V=800.0 PL=0
MOVL C00634 V=800.0 PL=0
MOVL C00635 V=800.0 PL=0
MOVL C00636 V=800.0 PL=0
MOVL C00637 V=800.0 PL=0
MOVL C00638 V=800.0 PL=0
MOVL C00639 V=800.0 PL=0
MOVL C00640 V=800.0 PL=0
MOVL C00641 V=800.0 PL=0
MOVL C00642 V=800.0 PL=0
MOVL C00643 V=800.0 PL=0
MOVL C00644 V=800.0 PL=0
MOVL C00645 V=800.0 PL=0
MOVL C00646 V=800.0 PL=0
MOVL C00647 V=800.0 PL=0
MOVL C00648 V=800.0 PL=0
MOVL C00649 V=800.0 PL=0
MOVL C00650 V=800.0 PL=0
MOVL C00651 V=800.0 PL=0
MOVL C00652 V=800.0 PL=0
MOVL C00653 V=800.0 PL=0
MOVL C00654 V=800.0 PL=0
MOVL C00655 V=800.0 PL=0
MOVL C00656 V=800.0 PL=0
MOVL C00657 V=800.0 PL=0
MOVL C00658 V=800.0 PL=0
MOVL C00659 V=800.0 PL=0
MOVL C00660 V=800.0 PL=0
MOVL C00661 V=800.0 PL=0
MOVL C00662 V=800.0 PL=0
MOVL C00663 V=800.0 PL=0
MOVL C00664 V=800.0 PL=0
MOVL C00665 V=800.0 PL=0
MOVL C00666 V=800.0 PL=0
MOVL C00667 V=800.0 PL=0
MOVL C00668 V=800.0 PL=0
MOVL C00669 V=800.0 PL=0
MOVL C00670 V=800.0 PL=0
MOVL C00671 V=800.0 PL=0
MOVL C00672 V=800.0 PL=0
MOVL C00673 V=800.0 PL=0
MOVL C00674 V=800.0 PL=0
MOVL C00675 V=800.0 PL=0
MOVL C00676 V=800.0 PL=0
MOVL C00677 V=800.0 PL=0
MOVL C00678 V=800.0 PL=0
MOVL C00679 V=800.0 PL=0
MOVL C00680 V=800.0 PL=0
MOVL C00681 V=800.0 PL=0
MOVL C00682 V=800.0 PL=0
MOVL C00683 V=800.0 PL=0
MOVL C00684 V=800.0 PL=0
MOVL C00685 V=800.0 PL=0
MOVL C00686 V=800.0 PL=0
MOVL C00687 V=800.0 PL=0
MOVL C00688 V=800.0 PL=0
MOVL C00689 V=800.0 PL=0
MOVL C00690 V=800.0 PL=0
MOVL C00691 V=800.0 PL=0
MOVL C00692 V=800.0 PL=0
MOVL C00693 V=800.0 PL=0
MOVL C00694 V=800.0 PL=0
MOVL C00695 V=800.0 PL=0
MOVL C00696 V=800.0 PL=0
MOVL C00697 V=800.0 PL=0
MOVL C00698 V=800.0 PL=0
MOVL C00699 V=800.0 PL=0
MOVL C00700 V=800.0 PL=0
MOVL C00701 V=800.0 PL=0
MOVL C00702 V=800.0 PL=0
MOVL C00703 V=800.0 PL=0
MOVL C00704 V=800.0 PL=0
MOVL C00705 V=800.0 PL=0
MOVL C00706 V=800.0 PL=0
MOVL C00707 V=800.0 PL=0
MOVL C00708 V=800.0 PL=0
MOVL C00709 V=800.0 PL=0
MOVL C00710 V=800.0 PL=0
MOVL C00711 V=800.0 PL=0
MOVL C00712 V=800.0 PL=0
MOVL C00713 V=800.0 PL=0
MOVL C00714 V=800.0 PL=0
MOVL C00715 V=800.0 PL=0
MOVL C00716 V=800.0 PL=0
MOVL C00717 V=800.0 PL=0
MOVL C00718 V=800.0 PL=0
MOVL C00719 V=800.0 PL=0
MOVL C00720 V=800.0 PL=0
MOVL C00721 V=800.0 PL=0
MOVL C00722 V=800.0 PL=0
MOVL C00723 V=800.0 PL=0
MOVL C00724 V=800.0 PL=0
MOVL C00725 V=800.0 PL=0
MOVL C00726 V=800.0 PL=0
MOVL C00727 V=800.0 PL=0
MOVL C00728 V=800.0 PL=0
MOVL C00729 V=800.0 PL=0
MOVL C00730 V=800.0 PL=0
MOVL C00731 V=800.0 PL=0
MOVL C00732 V=800.0 PL=0
MOVL C00733 V=800.0 PL=0
MOVL C00734 V=800.0 PL=0
MOVL C00735 V=800.0 PL=0
MOVL C00736 V=800.0 PL=0
MOVL C00737 V=800.0 PL=0
MOVL C00738 V=800.0 PL=0
MOVL C00739 V=800.0 PL=0
MOVL C00740 V=800.0 PL=0
MOVL C00741 V=800.0 PL=0
MOVL C00742 V=800.0 PL=0
MOVL C00743 V=800.0 PL=0
MOVL C00744 V=800.0 PL=0
MOVL C00745 V=800.0 PL=0
MOVL C00746 V=800.0 PL=0
MOVL C00747 V=800.0 PL=0
MOVL C00748 V=800.0 PL=0
MOVL C00749 V=800.0 PL=0
MOVL C00750 V=800.0 PL=0
MOVL C00751 V=800.0 PL=0
MOVL C00752 V=800.0 PL=0
MOVL C00753 V=800.0 PL=0
MOVL C00754 V=800.0 PL=0
MOVL C00755 V=800.0 PL=0
MOVL C00756 V=800.0 PL=0
MOVL C00757 V=800.0 PL=0
MOVL C00758 V=800.0 PL=0
MOVL C00759 V=800.0 PL=0
MOVL C00760 V=800.0 PL=0
MOVL C00761 V=800.0 PL=0
MOVL C00762 V=800.0 PL=0
MOVL C00763 V=800.0 PL=0
MOVL C00764 V=800.0 PL=0
MOVL C00765 V=800.0 PL=0
MOVL C00766 V=800.0 PL=0
MOVL C00767 V=800.0 PL=0
MOVL C00768 V=800.0 PL=0
MOVL C00769 V=800.0 PL=0
MOVL C00770 V=800.0 PL=0
MOVL C00771 V=800.0 PL=0
MOVL C00772 V=800.0 PL=0
MOVL C00773 V=800.0 PL=0
MOVL C00774 V=800.0 PL=0
MOVL C00775 V=800.0 PL=0
MOVL C00776 V=800.0 PL=0
MOVL C00777 V=800.0 PL=0
MOVL C00778 V=800.0 PL=0
MOVL C00779 V=800.0 PL=0
MOVL C00780 V=800.0 PL=0
MOVL C00781 V=800.0 PL=0
MOVL C00782 V=800.0 PL=0
MOVL C00783 V=800.0 PL=0
MOVL C00784 V=800.0 PL=0
MOVL C00785 V=800.0 PL=0
MOVL C00786 V=800.0 PL=0
MOVL C00787 V=800.0 PL=0
MOVL C00788 V=800.0 PL=0
MOVL C00789 V=800.0 PL=0
MOVL C00790 V=800.0 PL=0
MOVL C00791 V=800.0 PL=0
MOVL C00792 V=800.0 PL=0
MOVL C00793 V=800.0 PL=0
MOVL C00794 V=800.0 PL=0
MOVL C00795 V=800.0 PL=0
MOVL C00796 V=800.0 PL=0
MOVL C00797 V=800.0 PL=0
MOVL C00798 V=800.0 PL=0
MOVL C00799 V=800.0 PL=0
MOVL C00800 V=800.0 PL=0
MOVL C00801 V=800.0 PL=0
MOVL C00802 V=800.0 PL=0
MOVL C00803 V=800.0 PL=0
MOVL C00804 V=800.0 PL=0
MOVL C00805 V=800.0 PL=0
MOVL C00806 V=800.0 PL=0
MOVL C00807 V=800.0 PL=0
MOVL C00808 V=800.0 PL=0
MOVL C00809 V=800.0 PL=0
MOVL C00810 V=800.0 PL=0
MOVL C00811 V=800.0 PL=0
MOVL C00812 V=800.0 PL=0
MOVL C00813 V=800.0 PL=0
MOVL C00814 V=800.0 PL=0
MOVL C00815 V=800.0 PL=0
MOVL C00816 V=800.0 PL=0
MOVL C00817 V=800.0 PL=0
MOVL C00818 V=800.0 PL=0
MOVL C00819 V=800.0 PL=0
MOVL C00820 V=800.0 PL=0
MOVL C00821 V=800.0 PL=0
MOVL C00822 V=800.0 PL=0
MOVL C00823 V=800.0 PL=0
MOVL C00824 V=800.0 PL=0
MOVL C00825 V=800.0 PL=0
MOVL C00826 V=800.0 PL=0
MOVL C00827 V=800.0 PL=0
MOVL C00828 V=800.0 PL=0
MOVL C00829 V=800.0 PL=0
MOVL C00830 V=800.0 PL=0
MOVL C00831 V=800.0 PL=0
MOVL C00832 V=800.0 PL=0
MOVL C00833 V=800.0 PL=0
MOVL C00834 V=800.0 PL=0
MOVL C00835 V=800.0 PL=0
MOVL C00836 V=800.0 PL=0
MOVL C00837 V=800.0 PL=0
MOVL C00838 V=800.0 PL=0
MOVL C00839 V=800.0 PL=0
MOVL C00840 V=800.0 PL=0
MOVL C00841 V=800.0 PL=0
MOVL C00842 V=800.0 PL=0
MOVL C00843 V=800.0 PL=0
MOVL C00844 V=800.0 PL=0
MOVL C00845 V=800.0 PL=0
MOVL C00846 V=800.0 PL=0
MOVL C00847 V=800.0 PL=0
MOVL C00848 V=800.0 PL=0
MOVL C00849 V=800.0 PL=0
MOVL C00850 V=800.0 PL=0
MOVL C00851 V=800.0 PL=0
MOVL C00852 V=800.0 PL=0
MOVL C00853 V=800.0 PL=0
MOVL C00854 V=800.0 PL=0
MOVL C00855 V=800.0 PL=0
MOVL C00856 V=800.0 PL=0
MOVL C00857 V=800.0 PL=0
MOVL C00858 V=800.0 PL=0
MOVL C00859 V=800.0 PL=0
MOVL C00860 V=800.0 PL=0
MOVL C00861 V=800.0 PL=0
MOVL C00862 V=800.0 PL=0
MOVL C00863 V=800.0 PL=0
MOVL C00864 V=800.0 PL=0
MOVL C00865 V=800.0 PL=0
MOVL C00866 V=800.0 PL=0
MOVL C00867 V=800.0 PL=0
MOVL C00868 V=800.0 PL=0
MOVL C00869 V=800.0 PL=0
MOVL C00870 V=800.0 PL=0
MOVL C00871 V=800.0 PL=0
MOVL C00872 V=800.0 PL=0
MOVL C00873 V=800.0 PL=0
MOVL C00874 V=800.0 PL=0
MOVL C00875 V=800.0 PL=0
MOVL C00876 V=800.0 PL=0
MOVL C00877 V=800.0 PL=0
MOVL C00878 V=800.0 PL=0
MOVL C00879 V=800.0 PL=0
MOVL C00880 V=800.0 PL=0
MOVL C00881 V=800.0 PL=0
MOVL C00882 V=800.0 PL=0
MOVL C00883 V=800.0 PL=0
MOVL C00884 V=800.0 PL=0
MOVL C00885 V=800.0 PL=0
MOVL C00886 V=800.0 PL=0
MOVL C00887 V=800.0 PL=0
MOVL C00888 V=800.0 PL=0
MOVL C00889 V=800.0 PL=0
MOVL C00890 V=800.0 PL=0
MOVL C00891 V=800.0 PL=0
MOVL C00892 V=800.0 PL=0
MOVL C00893 V=800.0 PL=0
MOVL C00894 V=800.0 PL=0
MOVL C00895 V=800.0 PL=0
MOVL C00896 V=800.0 PL=0
MOVL C00897 V=800.0 PL=0
MOVL C00898 V=800.0 PL=0
MOVL C00899 V=800.0 PL=0
MOVL C00900 V=800.0 PL=0
MOVL C00901 V=800.0 PL=0
MOVL C00902 V=800.0 PL=0
MOVL C00903 V=800.0 PL=0
MOVL C00904 V=800.0 PL=0
MOVL C00905 V=800.0 PL=0
MOVL C00906 V=800.0 PL=0
MOVL C00907 V=800.0 PL=0
MOVL C00908 V=800.0 PL=0
MOVL C00909 V=800.0 PL=0
MOVL C00910 V=800.0 PL=0
MOVL C00911 V=800.0 PL=0
MOVL C00912 V=800.0 PL=0
MOVL C00913 V=800.0 PL=0
MOVL C00914 V=800.0 PL=0
MOVL C00915 V=800.0 PL=0
MOVL C00916 V=800.0 PL=0
MOVL C00917 V=800.0 PL=0
MOVL C00918 V=800.0 PL=0
MOVL C00919 V=800.0 PL=0
MOVL C00920 V=800.0 PL=0
MOVL C00921 V=800.0 PL=0
MOVL C00922 V=800.0 PL=0
MOVL C00923 V=800.0 PL=0
MOVL C00924 V=800.0 PL=0
MOVL C00925 V=800.0 PL=0
MOVL C00926 V=800.0 PL=0
MOVL C00927 V=800.0 PL=0
MOVL C00928 V=800.0 PL=0
MOVL C00929 V=800.0 PL=0
MOVL C00930 V=800.0 PL=0
MOVL C00931 V=800.0 PL=0
MOVL C00932 V=800.0 PL=0
MOVL C00933 V=800.0 PL=0
MOVL C00934 V=800.0 PL=0
MOVL C00935 V=800.0 PL=0
MOVL C00936 V=800.0 PL=0
MOVL C00937 V=800.0 PL=0
MOVL C00938 V=800.0 PL=0
MOVL C00939 V=800.0 PL=0
MOVL C00940 V=800.0 PL=0
MOVL C00941 V=800.0 PL=0
MOVL C00942 V=800.0 PL=0
MOVL C00943 V=800.0 PL=0
MOVL C00944 V=800.0 PL=0
MOVL C00945 V=800.0 PL=0
MOVL C00946 V=800.0 PL=0
MOVL C00947 V=800.0 PL=0
MOVL C00948 V=800.0 PL=0
MOVL C00949 V=800.0 PL=0
MOVL C00950 V=800.0 PL=0
MOVL C00951 V=800.0 PL=0
MOVL C00952 V=800.0 PL=0
MOVL C00953 V=800.0 PL=0
MOVL C00954 V=800.0 PL=0
MOVL C00955 V=800.0 PL=0
MOVL C00956 V=800.0 PL=0
MOVL C00957 V=800.0 PL=0
MOVL C00958 V=800.0 PL=0
MOVL C00959 V=800.0 PL=0
MOVL C00960 V=800.0 PL=0
MOVL C00961 V=800.0 PL=0
MOVL C00962 V=800.0 PL=0
MOVL C00963 V=800.0 PL=0
MOVL C00964 V=800.0 PL=0
MOVL C00965 V=800.0 PL=0
MOVL C00966 V=800.0 PL=0
MOVL C00967 V=800.0 PL=0
MOVL C00968 V=800.0 PL=0
MOVL C00969 V=800.0 PL=0
MOVL C00970 V=800.0 PL=0
MOVL C00971 V=800.0 PL=0
MOVL C00972 V=800.0 PL=0
MOVL C00973 V=800.0 PL=0
MOVL C00974 V=800.0 PL=0
MOVL C00975 V=800.0 PL=0
MOVL C00976 V=800.0 PL=0
MOVL C00977 V=800.0 PL=0
MOVL C00978 V=800.0 PL=0
MOVL C00979 V=800.0 PL=0
MOVL C00980 V=800.0 PL=0
MOVL C00981 V=800.0 PL=0
MOVL C00982 V=800.0 PL=0
MOVL C00983 V=800.0 PL=0
MOVL C00984 V=800.0 PL=0
MOVL C00985 V=800.0 PL=0
MOVL C00986 V=800.0 PL=0
MOVL C00987 V=800.0 PL=0
MOVL C00988 V=800.0 PL=0
MOVL C00989 V=800.0 PL=0
MOVL C00990 V=800.0 PL=0
MOVL C00991 V=800.0 PL=0
MOVL C00992 V=800.0 PL=0
MOVL C00993 V=800.0 PL=0
MOVL C00994 V=800.0 PL=0
MOVL C00995 V=800.0 PL=0
MOVL C00996 V=800.0 PL=0
MOVL C00997 V=800.0 PL=0
MOVL C00998 V=800.0 PL=0
MOVL C00999 V=800.0 PL=0
MOVL C01000 V=800.0 PL=0
MOVL C01001 V=800.0 PL=0
MOVL C01002 V=800.0 PL=0
MOVL C01003 V=800.0 PL=0
MOVL C01004 V=800.0 PL=0
MOVL C01005 V=800.0 PL=0
MOVL C01006 V=800.0 PL=0
MOVL C01007 V=800.0 PL=0
MOVL C01008 V=800.0 PL=0
MOVL C01009 V=800.0 PL=0
MOVL C01010 V=800.0 PL=0
MOVL C01011 V=800.0 PL=0
MOVL C01012 V=800.0 PL=0
MOVL C01013 V=800.0 PL=0
MOVL C01014 V=800.0 PL=0
MOVL C01015 V=800.0 PL=0
MOVL C01016 V=800.0 PL=0
MOVL C01017 V=800.0 PL=0
MOVL C01018 V=800.0 PL=0
MOVL C01019 V=800.0 PL=0
MOVL C01020 V=800.0 PL=0
MOVL C01021 V=800.0 PL=0
MOVL C01022 V=800.0 PL=0
MOVL C01023 V=800.0 PL=0
MOVL C01024 V=800.0 PL=0
MOVL C01025 V=800.0 PL=0
MOVL C01026 V=800.0 PL=0
MOVL C01027 V=800.0 PL=0
MOVL C01028 V=800.0 PL=0
MOVL C01029 V=800.0 PL=0
MOVL C01030 V=800.0 PL=0
MOVL C01031 V=800.0 PL=0
MOVL C01032 V=800.0 PL=0
MOVL C01033 V=800.0 PL=0
MOVL C01034 V=800.0 PL=0
MOVL C01035 V=800.0 PL=0
MOVL C01036 V=800.0 PL=0
MOVL C01037 V=800.0 PL=0
MOVL C01038 V=800.0 PL=0
MOVL C01039 V=800.0 PL=0
MOVL C01040 V=800.0 PL=0
MOVL C01041 V=800.0 PL=0
MOVL C01042 V=800.0 PL=0
MOVL C01043 V=800.0 PL=0
MOVL C01044 V=800.0 PL=0
MOVL C01045 V=800.0 PL=0
MOVL C01046 V=800.0 PL=0
MOVL C01047 V=800.0 PL=0
MOVL C01048 V=800.0 PL=0
MOVL C01049 V=800.0 PL=0
MOVL C01050 V=800.0 PL=0
MOVL C01051 V=800.0 PL=0
MOVL C01052 V=800.0 PL=0
MOVL C01053 V=800.0 PL=0
MOVL C01054 V=800.0 PL=0
MOVL C01055 V=800.0 PL=0
MOVL C01056 V=800.0 PL=0
MOVL C01057 V=800.0 PL=0
MOVL C01058 V=800.0 PL=0
MOVL C01059 V=800.0 PL=0
MOVL C01060 V=800.0 PL=0
MOVL C01061 V=800.0 PL=0
MOVL C01062 V=800.0 PL=0
MOVL C01063 V=800.0 PL=0
MOVL C01064 V=800.0 PL=0
MOVL C01065 V=800.0 PL=0
MOVL C01066 V=800.0 PL=0
MOVL C01067 V=800.0 PL=0
MOVL C01068 V=800.0 PL=0
MOVL C01069 V=800.0 PL=0
MOVL C01070 V=800.0 PL=0
MOVL C01071 V=800.0 PL=0
MOVL C01072 V=800.0 PL=0
MOVL C01073 V=800.0 PL=0
MOVL C01074 V=800.0 PL=0
MOVL C01075 V=800.0 PL=0
MOVL C01076 V=800.0 PL=0
MOVL C01077 V=800.0 PL=0
MOVL C01078 V=800.0 PL=0
MOVL C01079 V=800.0 PL=0
MOVL C01080 V=800.0 PL=0
MOVL C01081 V=800.0 PL=0
MOVL C01082 V=800.0 PL=0
MOVL C01083 V=800.0 PL=0
MOVL C01084 V=800.0 PL=0
MOVL C01085 V=800.0 PL=0
MOVL C01086 V=800.0 PL=0
MOVL C01087 V=800.0 PL=0
MOVL C01088 V=800.0 PL=0
MOVL C01089 V=800.0 PL=0
MOVL C01090 V=800.0 PL=0
MOVL C01091 V=800.0 PL=0
MOVL C01092 V=800.0 PL=0
MOVL C01093 V=800.0 PL=0
MOVL C01094 V=800.0 PL=0
MOVL C01095 V=800.0 PL=0
MOVL C01096 V=800.0 PL=0
MOVL C01097 V=800.0 PL=0
MOVL C01098 V=800.0 PL=0
MOVL C01099 V=800.0 PL=0
MOVL C01100 V=800.0 PL=0
MOVL C01101 V=800.0 PL=0
MOVL C01102 V=800.0 PL=0
MOVL C01103 V=800.0 PL=0
MOVL C01104 V=800.0 PL=0
MOVL C01105 V=800.0 PL=0
MOVL C01106 V=800.0 PL=0
MOVL C01107 V=800.0 PL=0
MOVL C01108 V=800.0 PL=0
MOVL C01109 V=800.0 PL=0
MOVL C01110 V=800.0 PL=0
MOVL C01111 V=800.0 PL=0
MOVL C01112 V=800.0 PL=0
MOVL C01113 V=800.0 PL=0
MOVL C01114 V=800.0 PL=0
MOVL C01115 V=800.0 PL=0
MOVL C01116 V=800.0 PL=0
MOVL C01117 V=800.0 PL=0
MOVL C01118 V=800.0 PL=0
MOVL C01119 V=800.0 PL=0
MOVL C01120 V=800.0 PL=0
MOVL C01121 V=800.0 PL=0
MOVL C01122 V=800.0 PL=0
MOVL C01123 V=800.0 PL=0
MOVL C01124 V=800.0 PL=0
MOVL C01125 V=800.0 PL=0
MOVL C01126 V=800.0 PL=0
MOVL C01127 V=800.0 PL=0
MOVL C01128 V=800.0 PL=0
MOVL C01129 V=800.0 PL=0
MOVL C01130 V=800.0 PL=0
MOVL C01131 V=800.0 PL=0
MOVL C01132 V=800.0 PL=0
MOVL C01133 V=800.0 PL=0
MOVL C01134 V=800.0 PL=0
MOVL C01135 V=800.0 PL=0
MOVL C01136 V=800.0 PL=0
MOVL C01137 V=800.0 PL=0
MOVL C01138 V=800.0 PL=0
MOVL C01139 V=800.0 PL=0
MOVL C01140 V=800.0 PL=0
MOVL C01141 V=800.0 PL=0
MOVL C01142 V=800.0 PL=0
MOVL C01143 V=800.0 PL=0
MOVL C01144 V=800.0 PL=0
MOVL C01145 V=800.0 PL=0
MOVL C01146 V=800.0 PL=0
MOVL C01147 V=800.0 PL=0
MOVL C01148 V=800.0 PL=0
MOVL C01149 V=800.0 PL=0
MOVL C01150 V=800.0 PL=0
MOVL C01151 V=800.0 PL=0
MOVL C01152 V=800.0 PL=0
MOVL C01153 V=800.0 PL=0
MOVL C01154 V=800.0 PL=0
MOVL C01155 V=800.0 PL=0
MOVL C01156 V=800.0 PL=0
MOVL C01157 V=800.0 PL=0
MOVL C01158 V=800.0 PL=0
MOVL C01159 V=800.0 PL=0
MOVL C01160 V=800.0 PL=0
MOVL C01161 V=800.0 PL=0
MOVL C01162 V=800.0 PL=0
MOVL C01163 V=800.0 PL=0
MOVL C01164 V=800.0 PL=0
MOVL C01165 V=800.0 PL=0
MOVL C01166 V=800.0 PL=0
MOVL C01167 V=800.0 PL=0
MOVL C01168 V=800.0 PL=0
MOVL C01169 V=800.0 PL=0
MOVL C01170 V=800.0 PL=0
MOVL C01171 V=800.0 PL=0
MOVL C01172 V=800.0 PL=0
MOVL C01173 V=800.0 PL=0
MOVL C01174 V=800.0 PL=0
MOVL C01175 V=800.0 PL=0
MOVL C01176 V=800.0 PL=0
MOVL C01177 V=800.0 PL=0
MOVL C01178 V=800.0 PL=0
MOVL C01179 V=800.0 PL=0
MOVL C01180 V=800.0 PL=0
MOVL C01181 V=800.0 PL=0
MOVL C01182 V=800.0 PL=0
MOVL C01183 V=800.0 PL=0
MOVL C01184 V=800.0 PL=0
MOVL C01185 V=800.0 PL=0
MOVL C01186 V=800.0 PL=0
MOVL C01187 V=800.0 PL=0
MOVL C01188 V=800.0 PL=0
MOVL C01189 V=800.0 PL=0
MOVL C01190 V=800.0 PL=0
MOVL C01191 V=800.0 PL=0
MOVL C01192 V=800.0 PL=0
MOVL C01193 V=800.0 PL=0
MOVL C01194 V=800.0 PL=0
MOVL C01195 V=800.0 PL=0
MOVL C01196 V=800.0 PL=0
MOVL C01197 V=800.0 PL=0
MOVL C01198 V=800.0 PL=0
MOVL C01199 V=800.0 PL=0
MOVL C01200 V=800.0 PL=0
MOVL C01201 V=800.0 PL=0
MOVL C01202 V=800.0 PL=0
MOVL C01203 V=800.0 PL=0
MOVL C01204 V=800.0 PL=0
MOVL C01205 V=800.0 PL=0
MOVL C01206 V=800.0 PL=0
MOVL C01207 V=800.0 PL=0
MOVL C01208 V=800.0 PL=0
MOVL C01209 V=800.0 PL=0
MOVL C01210 V=800.0 PL=0
MOVL C01211 V=800.0 PL=0
MOVL C01212 V=800.0 PL=0
MOVL C01213 V=800.0 PL=0
MOVL C01214 V=800.0 PL=0
MOVL C01215 V=800.0 PL=0
MOVL C01216 V=800.0 PL=0
MOVL C01217 V=800.0 PL=0
MOVL C01218 V=800.0 PL=0
MOVL C01219 V=800.0 PL=0
MOVL C01220 V=800.0 PL=0
MOVL C01221 V=800.0 PL=0
MOVL C01222 V=800.0 PL=0
MOVL C01223 V=800.0 PL=0
MOVL C01224 V=800.0 PL=0
MOVL C01225 V=800.0 PL=0
MOVL C01226 V=800.0 PL=0
MOVL C01227 V=800.0 PL=0
MOVL C01228 V=800.0 PL=0
MOVL C01229 V=800.0 PL=0
MOVL C01230 V=800.0 PL=0
MOVL C01231 V=800.0 PL=0
MOVL C01232 V=800.0 PL=0
MOVL C01233 V=800.0 PL=0
MOVL C01234 V=800.0 PL=0
MOVL C01235 V=800.0 PL=0
MOVL C01236 V=800.0 PL=0
MOVL C01237 V=800.0 PL=0
MOVL C01238 V=800.0 PL=0
MOVL C01239 V=800.0 PL=0
MOVL C01240 V=800.0 PL=0
MOVL C01241 V=800.0 PL=0
MOVL C01242 V=800.0 PL=0
MOVL C01243 V=800.0 PL=0
MOVL C01244 V=800.0 PL=0
MOVL C01245 V=800.0 PL=0
MOVL C01246 V=800.0 PL=0
MOVL C01247 V=800.0 PL=0
MOVL C01248 V=800.0 PL=0
MOVL C01249 V=800.0 PL=0
MOVL C01250 V=800.0 PL=0
MOVL C01251 V=800.0 PL=0
MOVL C01252 V=800.0 PL=0
MOVL C01253 V=800.0 PL=0
MOVL C01254 V=800.0 PL=0
MOVL C01255 V=800.0 PL=0
MOVL C01256 V=800.0 PL=0
MOVL C01257 V=800.0 PL=0
MOVL C01258 V=800.0 PL=0
MOVL C01259 V=800.0 PL=0
MOVL C01260 V=800.0 PL=0
MOVL C01261 V=800.0 PL=0
MOVL C01262 V=800.0 PL=0
MOVL C01263 V=800.0 PL=0
MOVL C01264 V=800.0 PL=0
MOVL C01265 V=800.0 PL=0
MOVL C01266 V=800.0 PL=0
MOVL C01267 V=800.0 PL=0
MOVL C01268 V=800.0 PL=0
MOVL C01269 V=800.0 PL=0
MOVL C01270 V=800.0 PL=0
MOVL C01271 V=800.0 PL=0
MOVL C01272 V=800.0 PL=0
MOVL C01273 V=800.0 PL=0
MOVL C01274 V=800.0 PL=0
MOVL C01275 V=800.0 PL=0
MOVL C01276 V=800.0 PL=0
MOVL C01277 V=800.0 PL=0
MOVL C01278 V=800.0 PL=0
MOVL C01279 V=800.0 PL=0
MOVL C01280 V=800.0 PL=0
MOVL C01281 V=800.0 PL=0
MOVL C01282 V=800.0 PL=0
MOVL C01283 V=800.0 PL=0
MOVL C01284 V=800.0 PL=0
MOVL C01285 V=800.0 PL=0
MOVL C01286 V=800.0 PL=0
MOVL C01287 V=800.0 PL=0
MOVL C01288 V=800.0 PL=0
MOVL C01289 V=800.0 PL=0
MOVL C01290 V=800.0 PL=0
MOVL C01291 V=800.0 PL=0
MOVL C01292 V=800.0 PL=0
MOVL C01293 V=800.0 PL=0
MOVL C01294 V=800.0 PL=0
MOVL C01295 V=800.0 PL=0
MOVL C01296 V=800.0 PL=0
MOVL C01297 V=800.0 PL=0
MOVL C01298 V=800.0 PL=0
MOVL C01299 V=800.0 PL=0
MOVL C01300 V=800.0 PL=0
MOVL C01301 V=800.0 PL=0
MOVL C01302 V=800.0 PL=0
MOVL C01303 V=800.0 PL=0
MOVL C01304 V=800.0 PL=0
MOVL C01305 V=800.0 PL=0
MOVL C01306 V=800.0 PL=0
MOVL C01307 V=800.0 PL=0
MOVL C01308 V=800.0 PL=0
MOVL C01309 V=800.0 PL=0
MOVL C01310 V=800.0 PL=0
MOVL C01311 V=800.0 PL=0
MOVL C01312 V=800.0 PL=0
MOVL C01313 V=800.0 PL=0
MOVL C01314 V=800.0 PL=0
MOVL C01315 V=800.0 PL=0
MOVL C01316 V=800.0 PL=0
MOVL C01317 V=800.0 PL=0
MOVL C01318 V=800.0 PL=0
MOVL C01319 V=800.0 PL=0
MOVL C01320 V=800.0 PL=0
MOVL C01321 V=800.0 PL=0
MOVL C01322 V=800.0 PL=0
MOVL C01323 V=800.0 PL=0
MOVL C01324 V=800.0 PL=0
MOVL C01325 V=800.0 PL=0
MOVL C01326 V=800.0 PL=0
MOVL C01327 V=800.0 PL=0
MOVL C01328 V=800.0 PL=0
MOVL C01329 V=800.0 PL=0
MOVL C01330 V=800.0 PL=0
MOVL C01331 V=800.0 PL=0
MOVL C01332 V=800.0 PL=0
MOVL C01333 V=800.0 PL=0
MOVL C01334 V=800.0 PL=0
MOVL C01335 V=800.0 PL=0
MOVL C01336 V=800.0 PL=0
MOVL C01337 V=800.0 PL=0
MOVL C01338 V=800.0 PL=0
MOVL C01339 V=800.0 PL=0
MOVL C01340 V=800.0 PL=0
MOVL C01341 V=800.0 PL=0
MOVL C01342 V=800.0 PL=0
MOVL C01343 V=800.0 PL=0
MOVL C01344 V=800.0 PL=0
MOVL C01345 V=800.0 PL=0
MOVL C01346 V=800.0 PL=0
MOVL C01347 V=800.0 PL=0
MOVL C01348 V=800.0 PL=0
MOVL C01349 V=800.0 PL=0
MOVL C01350 V=800.0 PL=0
MOVL C01351 V=800.0 PL=0
MOVL C01352 V=800.0 PL=0
MOVL C01353 V=800.0 PL=0
MOVL C01354 V=800.0 PL=0
MOVL C01355 V=800.0 PL=0
MOVL C01356 V=800.0 PL=0
MOVL C01357 V=800.0 PL=0
MOVL C01358 V=800.0 PL=0
MOVL C01359 V=800.0 PL=0
MOVL C01360 V=800.0 PL=0
MOVL C01361 V=800.0 PL=0
MOVL C01362 V=800.0 PL=0
MOVL C01363 V=800.0 PL=0
MOVL C01364 V=800.0 PL=0
MOVL C01365 V=800.0 PL=0
MOVL C01366 V=800.0 PL=0
MOVL C01367 V=800.0 PL=0
MOVL C01368 V=800.0 PL=0
MOVL C01369 V=800.0 PL=0
MOVL C01370 V=800.0 PL=0
MOVL C01371 V=800.0 PL=0
MOVL C01372 V=800.0 PL=0
MOVL C01373 V=800.0 PL=0
MOVL C01374 V=800.0 PL=0
MOVL C01375 V=800.0 PL=0
MOVL C01376 V=800.0 PL=0
MOVL C01377 V=800.0 PL=0
MOVL C01378 V=800.0 PL=0
MOVL C01379 V=800.0 PL=0
MOVL C01380 V=800.0 PL=0
MOVL C01381 V=800.0 PL=0
MOVL C01382 V=800.0 PL=0
MOVL C01383 V=800.0 PL=0
MOVL C01384 V=800.0 PL=0
MOVL C01385 V=800.0 PL=0
MOVL C01386 V=800.0 PL=0
MOVL C01387 V=800.0 PL=0
MOVL C01388 V=800.0 PL=0
MOVL C01389 V=800.0 PL=0
MOVL C01390 V=800.0 PL=0
MOVL C01391 V=800.0 PL=0
MOVL C01392 V=800.0 PL=0
MOVL C01393 V=800.0 PL=0
MOVL C01394 V=800.0 PL=0
MOVL C01395 V=800.0 PL=0
MOVL C01396 V=800.0 PL=0
MOVL C01397 V=800.0 PL=0
MOVL C01398 V=800.0 PL=0
MOVL C01399 V=800.0 PL=0
MOVL C01400 V=800.0 PL=0
MOVL C01401 V=800.0 PL=0
MOVL C01402 V=800.0 PL=0
MOVL C01403 V=800.0 PL=0
MOVL C01404 V=800.0 PL=0
MOVL C01405 V=800.0 PL=0
MOVL C01406 V=800.0 PL=0
MOVL C01407 V=800.0 PL=0
MOVL C01408 V=800.0 PL=0
MOVL C01409 V=800.0 PL=0
MOVL C01410 V=800.0 PL=0
MOVL C01411 V=800.0 PL=0
MOVL C01412 V=800.0 PL=0
MOVL C01413 V=800.0 PL=0
MOVL C01414 V=800.0 PL=0
MOVL C01415 V=800.0 PL=0
MOVL C01416 V=800.0 PL=0
MOVL C01417 V=800.0 PL=0
MOVL C01418 V=800.0 PL=0
MOVL C01419 V=800.0 PL=0
MOVL C01420 V=800.0 PL=0
MOVL C01421 V=800.0 PL=0
MOVL C01422 V=800.0 PL=0
MOVL C01423 V=800.0 PL=0
MOVL C01424 V=800.0 PL=0
MOVL C01425 V=800.0 PL=0
MOVL C01426 V=800.0 PL=0
MOVL C01427 V=800.0 PL=0
MOVL C01428 V=800.0 PL=0
MOVL C01429 V=800.0 PL=0
MOVL C01430 V=800.0 PL=0
MOVL C01431 V=800.0 PL=0
MOVL C01432 V=800.0 PL=0
MOVL C01433 V=800.0 PL=0
MOVL C01434 V=800.0 PL=0
MOVL C01435 V=800.0 PL=0
MOVL C01436 V=800.0 PL=0
MOVL C01437 V=800.0 PL=0
MOVL C01438 V=800.0 PL=0
MOVL C01439 V=800.0 PL=0
MOVL C01440 V=800.0 PL=0
MOVL C01441 V=800.0 PL=0
MOVL C01442 V=800.0 PL=0
MOVL C01443 V=800.0 PL=0
MOVL C01444 V=800.0 PL=0
MOVL C01445 V=800.0 PL=0
MOVL C01446 V=800.0 PL=0
MOVL C01447 V=800.0 PL=0
MOVL C01448 V=800.0 PL=0
MOVL C01449 V=800.0 PL=0
MOVL C01450 V=800.0 PL=0
MOVL C01451 V=800.0 PL=0
MOVL C01452 V=800.0 PL=0
MOVL C01453 V=800.0 PL=0
MOVL C01454 V=800.0 PL=0
MOVL C01455 V=800.0 PL=0
MOVL C01456 V=800.0 PL=0
MOVL C01457 V=800.0 PL=0
MOVL C01458 V=800.0 PL=0
MOVL C01459 V=800.0 PL=0
MOVL C01460 V=800.0 PL=0
MOVL C01461 V=800.0 PL=0
MOVL C01462 V=800.0 PL=0
MOVL C01463 V=800.0 PL=0
MOVL C01464 V=800.0 PL=0
MOVL C01465 V=800.0 PL=0
MOVL C01466 V=800.0 PL=0
MOVL C01467 V=800.0 PL=0
MOVL C01468 V=800.0 PL=0
MOVL C01469 V=800.0 PL=0
MOVL C01470 V=800.0 PL=0
MOVL C01471 V=800.0 PL=0
MOVL C01472 V=800.0 PL=0
MOVL C01473 V=800.0 PL=0
MOVL C01474 V=800.0 PL=0
MOVL C01475 V=800.0 PL=0
MOVL C01476 V=800.0 PL=0
MOVL C01477 V=800.0 PL=0
MOVL C01478 V=800.0 PL=0
MOVL C01479 V=800.0 PL=0
MOVL C01480 V=800.0 PL=0
MOVL C01481 V=800.0 PL=0
MOVL C01482 V=800.0 PL=0
MOVL C01483 V=800.0 PL=0
MOVL C01484 V=800.0 PL=0
MOVL C01485 V=800.0 PL=0
MOVL C01486 V=800.0 PL=0
MOVL C01487 V=800.0 PL=0
MOVL C01488 V=800.0 PL=0
MOVL C01489 V=800.0 PL=0
MOVL C01490 V=800.0 PL=0
MOVL C01491 V=800.0 PL=0
MOVL C01492 V=800.0 PL=0
MOVL C01493 V=800.0 PL=0
MOVL C01494 V=800.0 PL=0
MOVL C01495 V=800.0 PL=0
MOVL C01496 V=800.0 PL=0
MOVL C01497 V=800.0 PL=0
MOVL C01498 V=800.0 PL=0
MOVL C01499 V=800.0 PL=0
MOVL C01500 V=800.0 PL=0
MOVL C01501 V=800.0 PL=0
MOVL C01502 V=800.0 PL=0
MOVL C01503 V=800.0 PL=0
MOVL C01504 V=800.0 PL=0
MOVL C01505 V=800.0 PL=0
MOVL C01506 V=800.0 PL=0
MOVL C01507 V=800.0 PL=0
MOVL C01508 V=800.0 PL=0
MOVL C01509 V=800.0 PL=0
MOVL C01510 V=800.0 PL=0
MOVL C01511 V=800.0 PL=0
MOVL C01512 V=800.0 PL=0
MOVL C01513 V=800.0 PL=0
MOVL C01514 V=800.0 PL=0
MOVL C01515 V=800.0 PL=0
MOVL C01516 V=800.0 PL=0
MOVL C01517 V=800.0 PL=0
MOVL C01518 V=800.0 PL=0
MOVL C01519 V=800.0 PL=0
MOVL C01520 V=800.0 PL=0
MOVL C01521 V=800.0 PL=0
MOVL C01522 V=800.0 PL=0
MOVL C01523 V=800.0 PL=0
MOVL C01524 V=800.0 PL=0
MOVL C01525 V=800.0 PL=0
MOVL C01526 V=800.0 PL=0
MOVL C01527 V=800.0 PL=0
MOVL C01528 V=800.0 PL=0
MOVL C01529 V=800.0 PL=0
MOVL C01530 V=800.0 PL=0
MOVL C01531 V=800.0 PL=0
MOVL C01532 V=800.0 PL=0
MOVL C01533 V=800.0 PL=0
MOVL C01534 V=800.0 PL=0
MOVL C01535 V=800.0 PL=0
MOVL C01536 V=800.0 PL=0
MOVL C01537 V=800.0 PL=0
MOVL C01538 V=800.0 PL=0
MOVL C01539 V=800.0 PL=0
MOVL C01540 V=800.0 PL=0
MOVL C01541 V=800.0 PL=0
MOVL C01542 V=800.0 PL=0
MOVL C01543 V=800.0 PL=0
MOVL C01544 V=800.0 PL=0
MOVL C01545 V=800.0 PL=0
MOVL C01546 V=800.0 PL=0
MOVL C01547 V=800.0 PL=0
MOVL C01548 V=800.0 PL=0
MOVL C01549 V=800.0 PL=0
MOVL C01550 V=800.0 PL=0
MOVL C01551 V=800.0 PL=0
MOVL C01552 V=800.0 PL=0
MOVL C01553 V=800.0 PL=0
MOVL C01554 V=800.0 PL=0
MOVL C01555 V=800.0 PL=0
MOVL C01556 V=800.0 PL=0
MOVL C01557 V=800.0 PL=0
MOVL C01558 V=800.0 PL=0
MOVL C01559 V=800.0 PL=0
MOVL C01560 V=800.0 PL=0
MOVL C01561 V=800.0 PL=0
MOVL C01562 V=800.0 PL=0
MOVL C01563 V=800.0 PL=0
MOVL C01564 V=800.0 PL=0
MOVL C01565 V=800.0 PL=0
MOVL C01566 V=800.0 PL=0
MOVL C01567 V=800.0 PL=0
MOVL C01568 V=800.0 PL=0
MOVL C01569 V=800.0 PL=0
MOVL C01570 V=800.0 PL=0
MOVL C01571 V=800.0 PL=0
MOVL C01572 V=800.0 PL=0
MOVL C01573 V=800.0 PL=0
MOVL C01574 V=800.0 PL=0
MOVL C01575 V=800.0 PL=0
MOVL C01576 V=800.0 PL=0
MOVL C01577 V=800.0 PL=0
MOVL C01578 V=800.0 PL=0
MOVL C01579 V=800.0 PL=0
MOVL C01580 V=800.0 PL=0
MOVL C01581 V=800.0 PL=0
MOVL C01582 V=800.0 PL=0
MOVL C01583 V=800.0 PL=0
MOVL C01584 V=800.0 PL=0
MOVL C01585 V=800.0 PL=0
MOVL C01586 V=800.0 PL=0
MOVL C01587 V=800.0 PL=0
MOVL C01588 V=800.0 PL=0
MOVL C01589 V=800.0 PL=0
MOVL C01590 V=800.0 PL=0
MOVL C01591 V=800.0 PL=0
MOVL C01592 V=800.0 PL=0
MOVL C01593 V=800.0 PL=0
MOVL C01594 V=800.0 PL=0
MOVL C01595 V=800.0 PL=0
MOVL C01596 V=800.0 PL=0
MOVL C01597 V=800.0 PL=0
MOVL C01598 V=800.0 PL=0
MOVL C01599 V=800.0 PL=0
MOVL C01600 V=800.0 PL=0
MOVL C01601 V=800.0 PL=0
MOVL C01602 V=800.0 PL=0
MOVL C01603 V=800.0 PL=0
MOVL C01604 V=800.0 PL=0
MOVL C01605 V=800.0 PL=0
MOVL C01606 V=800.0 PL=0
MOVL C01607 V=800.0 PL=0
MOVL C01608 V=800.0 PL=0
MOVL C01609 V=800.0 PL=0
MOVL C01610 V=800.0 PL=0
MOVL C01611 V=800.0 PL=0
MOVL C01612 V=800.0 PL=0
MOVL C01613 V=800.0 PL=0
MOVL C01614 V=800.0 PL=0
MOVL C01615 V=800.0 PL=0
MOVL C01616 V=800.0 PL=0
MOVL C01617 V=800.0 PL=0
MOVL C01618 V=800.0 PL=0
MOVL C01619 V=800.0 PL=0
MOVL C01620 V=800.0 PL=0
MOVL C01621 V=800.0 PL=0
MOVL C01622 V=800.0 PL=0
MOVL C01623 V=800.0 PL=0
MOVL C01624 V=800.0 PL=0
MOVL C01625 V=800.0 PL=0
MOVL C01626 V=800.0 PL=0
MOVL C01627 V=800.0 PL=0
MOVL C01628 V=800.0 PL=0
MOVL C01629 V=800.0 PL=0
MOVL C01630 V=800.0 PL=0
MOVL C01631 V=800.0 PL=0
MOVL C01632 V=800.0 PL=0
MOVL C01633 V=800.0 PL=0
MOVL C01634 V=800.0 PL=0
MOVL C01635 V=800.0 PL=0
MOVL C01636 V=800.0 PL=0
MOVL C01637 V=800.0 PL=0
MOVL C01638 V=800.0 PL=0
MOVL C01639 V=800.0 PL=0
MOVL C01640 V=800.0 PL=0
MOVL C01641 V=800.0 PL=0
MOVL C01642 V=800.0 PL=0
MOVL C01643 V=800.0 PL=0
MOVL C01644 V=800.0 PL=0
MOVL C01645 V=800.0 PL=0
MOVL C01646 V=800.0 PL=0
MOVL C01647 V=800.0 PL=0
MOVL C01648 V=800.0 PL=0
MOVL C01649 V=800.0 PL=0
MOVL C01650 V=800.0 PL=0
MOVL C01651 V=800.0 PL=0
MOVL C01652 V=800.0 PL=0
MOVL C01653 V=800.0 PL=0
MOVL C01654 V=800.0 PL=0
MOVL C01655 V=800.0 PL=0
MOVL C01656 V=800.0 PL=0
MOVL C01657 V=800.0 PL=0
MOVL C01658 V=800.0 PL=0
MOVL C01659 V=800.0 PL=0
MOVL C01660 V=800.0 PL=0
MOVL C01661 V=800.0 PL=0
MOVL C01662 V=800.0 PL=0
MOVL C01663 V=800.0 PL=0
MOVL C01664 V=800.0 PL=0
MOVL C01665 V=800.0 PL=0
MOVL C01666 V=800.0 PL=0
MOVL C01667 V=800.0 PL=0
MOVL C01668 V=800.0 PL=0
MOVL C01669 V=800.0 PL=0
MOVL C01670 V=800.0 PL=0
MOVL C01671 V=800.0 PL=0
MOVL C01672 V=800.0 PL=0
MOVL C01673 V=800.0 PL=0
MOVL C01674 V=800.0 PL=0
MOVL C01675 V=800.0 PL=0
MOVL C01676 V=800.0 PL=0
MOVL C01677 V=800.0 PL=0
MOVL C01678 V=800.0 PL=0
MOVL C01679 V=800.0 PL=0
MOVL C01680 V=800.0 PL=0
MOVL C01681 V=800.0 PL=0
MOVL C01682 V=800.0 PL=0
MOVL C01683 V=800.0 PL=0
MOVL C01684 V=800.0 PL=0
MOVL C01685 V=800.0 PL=0
MOVL C01686 V=800.0 PL=0
MOVL C01687 V=800.0 PL=0
MOVL C01688 V=800.0 PL=0
MOVL C01689 V=800.0 PL=0
MOVL C01690 V=800.0 PL=0
MOVL C01691 V=800.0 PL=0
MOVL C01692 V=800.0 PL=0
MOVL C01693 V=800.0 PL=0
MOVL C01694 V=800.0 PL=0
MOVL C01695 V=800.0 PL=0
MOVL C01696 V=800.0 PL=0
MOVL C01697 V=800.0 PL=0
MOVL C01698 V=800.0 PL=0
MOVL C01699 V=800.0 PL=0
MOVL C01700 V=800.0 PL=0
MOVL C01701 V=800.0 PL=0
MOVL C01702 V=800.0 PL=0
MOVL C01703 V=800.0 PL=0
MOVL C01704 V=800.0 PL=0
MOVL C01705 V=800.0 PL=0
MOVL C01706 V=800.0 PL=0
MOVL C01707 V=800.0 PL=0
MOVL C01708 V=800.0 PL=0
MOVL C01709 V=800.0 PL=0
MOVL C01710 V=800.0 PL=0
MOVL C01711 V=800.0 PL=0
MOVL C01712 V=800.0 PL=0
MOVL C01713 V=800.0 PL=0
MOVL C01714 V=800.0 PL=0
MOVL C01715 V=800.0 PL=0
MOVL C01716 V=800.0 PL=0
MOVL C01717 V=800.0 PL=0
MOVL C01718 V=800.0 PL=0
MOVL C01719 V=800.0 PL=0
MOVL C01720 V=800.0 PL=0
MOVL C01721 V=800.0 PL=0
MOVL C01722 V=800.0 PL=0
MOVL C01723 V=800.0 PL=0
MOVL C01724 V=800.0 PL=0
MOVL C01725 V=800.0 PL=0
MOVL C01726 V=800.0 PL=0
MOVL C01727 V=800.0 PL=0
MOVL C01728 V=800.0 PL=0
MOVL C01729 V=800.0 PL=0
MOVL C01730 V=800.0 PL=0
MOVL C01731 V=800.0 PL=0
MOVL C01732 V=800.0 PL=0
MOVL C01733 V=800.0 PL=0
MOVL C01734 V=800.0 PL=0
MOVL C01735 V=800.0 PL=0
MOVL C01736 V=800.0 PL=0
MOVL C01737 V=800.0 PL=0
MOVL C01738 V=800.0 PL=0
MOVL C01739 V=800.0 PL=0
MOVL C01740 V=800.0 PL=0
MOVL C01741 V=800.0 PL=0
MOVL C01742 V=800.0 PL=0
MOVL C01743 V=800.0 PL=0
MOVL C01744 V=800.0 PL=0
MOVL C01745 V=800.0 PL=0
MOVL C01746 V=800.0 PL=0
MOVL C01747 V=800.0 PL=0
MOVL C01748 V=800.0 PL=0
MOVL C01749 V=800.0 PL=0
MOVL C01750 V=800.0 PL=0
MOVL C01751 V=800.0 PL=0
MOVL C01752 V=800.0 PL=0
MOVL C01753 V=800.0 PL=0
MOVL C01754 V=800.0 PL=0
MOVL C01755 V=800.0 PL=0
MOVL C01756 V=800.0 PL=0
MOVL C01757 V=800.0 PL=0
MOVL C01758 V=800.0 PL=0
MOVL C01759 V=800.0 PL=0
MOVL C01760 V=800.0 PL=0
MOVL C01761 V=800.0 PL=0
MOVL C01762 V=800.0 PL=0
MOVL C01763 V=800.0 PL=0
MOVL C01764 V=800.0 PL=0
MOVL C01765 V=800.0 PL=0
MOVL C01766 V=800.0 PL=0
MOVL C01767 V=800.0 PL=0
MOVL C01768 V=800.0 PL=0
MOVL C01769 V=800.0 PL=0
MOVL C01770 V=800.0 PL=0
MOVL C01771 V=800.0 PL=0
MOVL C01772 V=800.0 PL=0
MOVL C01773 V=800.0 PL=0
MOVL C01774 V=800.0 PL=0
MOVL C01775 V=800.0 PL=0
MOVL C01776 V=800.0 PL=0
MOVL C01777 V=800.0 PL=0
MOVL C01778 V=800.0 PL=0
MOVL C01779 V=800.0 PL=0
MOVL C01780 V=800.0 PL=0
MOVL C01781 V=800.0 PL=0
MOVL C01782 V=800.0 PL=0
MOVL C01783 V=800.0 PL=0
MOVL C01784 V=800.0 PL=0
MOVL C01785 V=800.0 PL=0
MOVL C01786 V=800.0 PL=0
MOVL C01787 V=800.0 PL=0
MOVL C01788 V=800.0 PL=0
MOVL C01789 V=800.0 PL=0
MOVL C01790 V=800.0 PL=0
MOVL C01791 V=800.0 PL=0
MOVL C01792 V=800.0 PL=0
MOVL C01793 V=800.0 PL=0
MOVL C01794 V=800.0 PL=0
MOVL C01795 V=800.0 PL=0
MOVL C01796 V=800.0 PL=0
MOVL C01797 V=800.0 PL=0
MOVL C01798 V=800.0 PL=0
MOVL C01799 V=800.0 PL=0
MOVL C01800 V=800.0 PL=0
MOVL C01801 V=800.0 PL=0
MOVL C01802 V=800.0 PL=0
MOVL C01803 V=800.0 PL=0
MOVL C01804 V=800.0 PL=0
MOVL C01805 V=800.0 PL=0
MOVL C01806 V=800.0 PL=0
MOVL C01807 V=800.0 PL=0
MOVL C01808 V=800.0 PL=0
MOVL C01809 V=800.0 PL=0
MOVL C01810 V=800.0 PL=0
MOVL C01811 V=800.0 PL=0
MOVL C01812 V=800.0 PL=0
MOVL C01813 V=800.0 PL=0
MOVL C01814 V=800.0 PL=0
MOVL C01815 V=800.0 PL=0
MOVL C01816 V=800.0 PL=0
MOVL C01817 V=800.0 PL=0
MOVL C01818 V=800.0 PL=0
MOVL C01819 V=800.0 PL=0
MOVL C01820 V=800.0 PL=0
MOVL C01821 V=800.0 PL=0
MOVL C01822 V=800.0 PL=0
MOVL C01823 V=800.0 PL=0
MOVL C01824 V=800.0 PL=0
MOVL C01825 V=800.0 PL=0
MOVL C01826 V=800.0 PL=0
MOVL C01827 V=800.0 PL=0
MOVL C01828 V=800.0 PL=0
MOVL C01829 V=800.0 PL=0
MOVL C01830 V=800.0 PL=0
MOVL C01831 V=800.0 PL=0
MOVL C01832 V=800.0 PL=0
MOVL C01833 V=800.0 PL=0
MOVL C01834 V=800.0 PL=0
MOVL C01835 V=800.0 PL=0
MOVL C01836 V=800.0 PL=0
MOVL C01837 V=800.0 PL=0
MOVL C01838 V=800.0 PL=0
MOVL C01839 V=800.0 PL=0
MOVL C01840 V=800.0 PL=0
MOVL C01841 V=800.0 PL=0
MOVL C01842 V=800.0 PL=0
MOVL C01843 V=800.0 PL=0
MOVL C01844 V=800.0 PL=0
MOVL C01845 V=800.0 PL=0
MOVL C01846 V=800.0 PL=0
MOVL C01847 V=800.0 PL=0
MOVL C01848 V=800.0 PL=0
MOVL C01849 V=800.0 PL=0
MOVL C01850 V=800.0 PL=0
MOVL C01851 V=800.0 PL=0
MOVL C01852 V=800.0 PL=0
MOVL C01853 V=800.0 PL=0
MOVL C01854 V=800.0 PL=0
MOVL C01855 V=800.0 PL=0
MOVL C01856 V=800.0 PL=0
MOVL C01857 V=800.0 PL=0
MOVL C01858 V=800.0 PL=0
MOVL C01859 V=800.0 PL=0
MOVL C01860 V=800.0 PL=0
MOVL C01861 V=800.0 PL=0
MOVL C01862 V=800.0 PL=0
MOVL C01863 V=800.0 PL=0
MOVL C01864 V=800.0 PL=0
MOVL C01865 V=800.0 PL=0
MOVL C01866 V=800.0 PL=0
MOVL C01867 V=800.0 PL=0
MOVL C01868 V=800.0 PL=0
MOVL C01869 V=800.0 PL=0
MOVL C01870 V=800.0 PL=0
MOVL C01871 V=800.0 PL=0
MOVL C01872 V=800.0 PL=0
MOVL C01873 V=800.0 PL=0
MOVL C01874 V=800.0 PL=0
MOVL C01875 V=800.0 PL=0
MOVL C01876 V=800.0 PL=0
MOVL C01877 V=800.0 PL=0
MOVL C01878 V=800.0 PL=0
MOVL C01879 V=800.0 PL=0
MOVL C01880 V=800.0 PL=0
MOVL C01881 V=800.0 PL=0
MOVL C01882 V=800.0 PL=0
MOVL C01883 V=800.0 PL=0
MOVL C01884 V=800.0 PL=0
MOVL C01885 V=800.0 PL=0
MOVL C01886 V=800.0 PL=0
MOVL C01887 V=800.0 PL=0
MOVL C01888 V=800.0 PL=0
MOVL C01889 V=800.0 PL=0
MOVL C01890 V=800.0 PL=0
MOVL C01891 V=800.0 PL=0
MOVL C01892 V=800.0 PL=0
MOVL C01893 V=800.0 PL=0
MOVL C01894 V=800.0 PL=0
MOVL C01895 V=800.0 PL=0
MOVL C01896 V=800.0 PL=0
MOVL C01897 V=800.0 PL=0
MOVL C01898 V=800.0 PL=0
MOVL C01899 V=800.0 PL=0
MOVL C01900 V=800.0 PL=0
MOVL C01901 V=800.0 PL=0
MOVL C01902 V=800.0 PL=0
MOVL C01903 V=800.0 PL=0
MOVL C01904 V=800.0 PL=0
MOVL C01905 V=800.0 PL=0
MOVL C01906 V=800.0 PL=0
MOVL C01907 V=800.0 PL=0
MOVL C01908 V=800.0 PL=0
MOVL C01909 V=800.0 PL=0
MOVL C01910 V=800.0 PL=0
MOVL C01911 V=800.0 PL=0
MOVL C01912 V=800.0 PL=0
MOVL C01913 V=800.0 PL=0
MOVL C01914 V=800.0 PL=0
MOVL C01915 V=800.0 PL=0
MOVL C01916 V=800.0 PL=0
MOVL C01917 V=800.0 PL=0
MOVL C01918 V=800.0 PL=0
MOVL C01919 V=800.0 PL=0
MOVL C01920 V=800.0 PL=0
MOVL C01921 V=800.0 PL=0
MOVL C01922 V=800.0 PL=0
MOVL C01923 V=800.0 PL=0
MOVL C01924 V=800.0 PL=0
MOVL C01925 V=800.0 PL=0
MOVL C01926 V=800.0 PL=0
MOVL C01927 V=800.0 PL=0
MOVL C01928 V=800.0 PL=0
MOVL C01929 V=800.0 PL=0
MOVL C01930 V=800.0 PL=0
MOVL C01931 V=800.0 PL=0
MOVL C01932 V=800.0 PL=0
MOVL C01933 V=800.0 PL=0
MOVL C01934 V=800.0 PL=0
MOVL C01935 V=800.0 PL=0
MOVL C01936 V=800.0 PL=0
MOVL C01937 V=800.0 PL=0
MOVL C01938 V=800.0 PL=0
MOVL C01939 V=800.0 PL=0
MOVL C01940 V=800.0 PL=0
MOVL C01941 V=800.0 PL=0
MOVL C01942 V=800.0 PL=0
MOVL C01943 V=800.0 PL=0
MOVL C01944 V=800.0 PL=0
MOVL C01945 V=800.0 PL=0
MOVL C01946 V=800.0 PL=0
MOVL C01947 V=800.0 PL=0
MOVL C01948 V=800.0 PL=0
MOVL C01949 V=800.0 PL=0
MOVL C01950 V=800.0 PL=0
MOVL C01951 V=800.0 PL=0
MOVL C01952 V=800.0 PL=0
MOVL C01953 V=800.0 PL=0
MOVL C01954 V=800.0 PL=0
MOVL C01955 V=800.0 PL=0
MOVL C01956 V=800.0 PL=0
MOVL C01957 V=800.0 PL=0
MOVL C01958 V=800.0 PL=0
MOVL C01959 V=800.0 PL=0
MOVL C01960 V=800.0 PL=0
MOVL C01961 V=800.0 PL=0
MOVL C01962 V=800.0 PL=0
MOVL C01963 V=800.0 PL=0
MOVL C01964 V=800.0 PL=0
MOVL C01965 V=800.0 PL=0
MOVL C01966 V=800.0 PL=0
MOVL C01967 V=800.0 PL=0
MOVL C01968 V=800.0 PL=0
MOVL C01969 V=800.0 PL=0
MOVL C01970 V=800.0 PL=0
MOVL C01971 V=800.0 PL=0
MOVL C01972 V=800.0 PL=0
MOVL C01973 V=800.0 PL=0
MOVL C01974 V=800.0 PL=0
MOVL C01975 V=800.0 PL=0
MOVL C01976 V=800.0 PL=0
MOVL C01977 V=800.0 PL=0
MOVL C01978 V=800.0 PL=0
MOVL C01979 V=800.0 PL=0
MOVL C01980 V=800.0 PL=0
MOVL C01981 V=800.0 PL=0
MOVL C01982 V=800.0 PL=0
MOVL C01983 V=800.0 PL=0
MOVL C01984 V=800.0 PL=0
MOVL C01985 V=800.0 PL=0
MOVL C01986 V=800.0 PL=0
MOVL C01987 V=800.0 PL=0
MOVL C01988 V=800.0 PL=0
MOVL C01989 V=800.0 PL=0
MOVL C01990 V=800.0 PL=0
MOVL C01991 V=800.0 PL=0
MOVL C01992 V=800.0 PL=0
MOVL C01993 V=800.0 PL=0
MOVL C01994 V=800.0 PL=0
MOVL C01995 V=800.0 PL=0
MOVL C01996 V=800.0 PL=0
MOVL C01997 V=800.0 PL=0
MOVL C01998 V=800.0 PL=0
MOVL C01999 V=800.0 PL=0
MOVL C02000 V=800.0 PL=0
MOVL C02001 V=800.0 PL=0
MOVL C02002 V=800.0 PL=0
MOVL C02003 V=800.0 PL=0
MOVL C02004 V=800.0 PL=0
MOVL C02005 V=800.0 PL=0
MOVL C02006 V=800.0 PL=0
MOVL C02007 V=800.0 PL=0
MOVL C02008 V=800.0 PL=0
MOVL C02009 V=800.0 PL=0
MOVL C02010 V=800.0 PL=0
MOVL C02011 V=800.0 PL=0
MOVL C02012 V=800.0 PL=0
MOVL C02013 V=800.0 PL=0
MOVL C02014 V=800.0 PL=0
MOVL C02015 V=800.0 PL=0
MOVL C02016 V=800.0 PL=0
MOVL C02017 V=800.0 PL=0
MOVL C02018 V=800.0 PL=0
MOVL C02019 V=800.0 PL=0
MOVL C02020 V=800.0 PL=0
MOVL C02021 V=800.0 PL=0
MOVL C02022 V=800.0 PL=0
MOVL C02023 V=800.0 PL=0
MOVL C02024 V=800.0 PL=0
MOVL C02025 V=800.0 PL=0
MOVL C02026 V=800.0 PL=0
MOVL C02027 V=800.0 PL=0
MOVL C02028 V=800.0 PL=0
MOVL C02029 V=800.0 PL=0
MOVL C02030 V=800.0 PL=0
MOVL C02031 V=800.0 PL=0
MOVL C02032 V=800.0 PL=0
MOVL C02033 V=800.0 PL=0
MOVL C02034 V=800.0 PL=0
MOVL C02035 V=800.0 PL=0
MOVL C02036 V=800.0 PL=0
MOVL C02037 V=800.0 PL=0
MOVL C02038 V=800.0 PL=0
MOVL C02039 V=800.0 PL=0
MOVL C02040 V=800.0 PL=0
MOVL C02041 V=800.0 PL=0
MOVL C02042 V=800.0 PL=0
MOVL C02043 V=800.0 PL=0
MOVL C02044 V=800.0 PL=0
MOVL C02045 V=800.0 PL=0
MOVL C02046 V=800.0 PL=0
MOVL C02047 V=800.0 PL=0
MOVL C02048 V=800.0 PL=0
MOVL C02049 V=800.0 PL=0
MOVL C02050 V=800.0 PL=0
MOVL C02051 V=800.0 PL=0
MOVL C02052 V=800.0 PL=0
MOVL C02053 V=800.0 PL=0
MOVL C02054 V=800.0 PL=0
MOVL C02055 V=800.0 PL=0
MOVL C02056 V=800.0 PL=0
MOVL C02057 V=800.0 PL=0
MOVL C02058 V=800.0 PL=0
MOVL C02059 V=800.0 PL=0
MOVL C02060 V=800.0 PL=0
MOVL C02061 V=800.0 PL=0
MOVL C02062 V=800.0 PL=0
MOVL C02063 V=800.0 PL=0
MOVL C02064 V=800.0 PL=0
MOVL C02065 V=800.0 PL=0
MOVL C02066 V=800.0 PL=0
MOVL C02067 V=800.0 PL=0
MOVL C02068 V=800.0 PL=0
MOVL C02069 V=800.0 PL=0
MOVL C02070 V=800.0 PL=0
MOVL C02071 V=800.0 PL=0
MOVL C02072 V=800.0 PL=0
MOVL C02073 V=800.0 PL=0
MOVL C02074 V=800.0 PL=0
MOVL C02075 V=800.0 PL=0
MOVL C02076 V=800.0 PL=0
MOVL C02077 V=800.0 PL=0
MOVL C02078 V=800.0 PL=0
MOVL C02079 V=800.0 PL=0
MOVL C02080 V=800.0 PL=0
MOVL C02081 V=800.0 PL=0
MOVL C02082 V=800.0 PL=0
MOVL C02083 V=800.0 PL=0
MOVL C02084 V=800.0 PL=0
MOVL C02085 V=800.0 PL=0
MOVL C02086 V=800.0 PL=0
MOVL C02087 V=800.0 PL=0
MOVL C02088 V=800.0 PL=0
MOVL C02089 V=800.0 PL=0
MOVL C02090 V=800.0 PL=0
MOVL C02091 V=800.0 PL=0
MOVL C02092 V=800.0 PL=0
MOVL C02093 V=800.0 PL=0
MOVL C02094 V=800.0 PL=0
MOVL C02095 V=800.0 PL=0
MOVL C02096 V=800.0 PL=0
MOVL C02097 V=800.0 PL=0
MOVL C02098 V=800.0 PL=0
MOVL C02099 V=800.0 PL=0
MOVL C02100 V=800.0 PL=0
MOVL C02101 V=800.0 PL=0
MOVL C02102 V=800.0 PL=0
MOVL C02103 V=800.0 PL=0
MOVL C02104 V=800.0 PL=0
MOVL C02105 V=800.0 PL=0
MOVL C02106 V=800.0 PL=0
MOVL C02107 V=800.0 PL=0
MOVL C02108 V=800.0 PL=0
MOVL C02109 V=800.0 PL=0
MOVL C02110 V=800.0 PL=0
MOVL C02111 V=800.0 PL=0
MOVL C02112 V=800.0 PL=0
MOVL C02113 V=800.0 PL=0
MOVL C02114 V=800.0 PL=0
MOVL C02115 V=800.0 PL=0
MOVL C02116 V=800.0 PL=0
MOVL C02117 V=800.0 PL=0
MOVL C02118 V=800.0 PL=0
MOVL C02119 V=800.0 PL=0
MOVL C02120 V=800.0 PL=0
MOVL C02121 V=800.0 PL=0
